(* CODESYS project rmthtc3library.library
   Company: RMTH GmbH
   Title: RMTH TC3 Library
   Placeholder: RMTH TC3 Library
   Version: 1.7

Project tree, tasks and I/O mapping:
  libraries: Tc2_Drive, * (Beckhoff Automation GmbH); Tc2_EtherCAT, * (Beckhoff Automation GmbH); Tc2_MC2, * (Beckhoff Automation GmbH); Tc2_MC2_Drive, * (Beckhoff Automation GmbH); Tc2_NC, * (Beckhoff Automation GmbH); Tc2_Standard, * (Beckhoff Automation GmbH); Tc2_System, * (Beckhoff Automation GmbH); Tc2_Utilities, * (Beckhoff Automation GmbH); Tc3_Interfaces, * (Beckhoff Automation GmbH); Tc3_Module, * (Beckhoff Automation GmbH)
  Configuration/
    Log/
      data type E_LoggingProvider
      data type E_LogLevel
      data type ST_LoggingConfig
    Motion/
      data type E_AxisType
      data type E_EncoderType
  Motion/
    AX5000Diag/
      Structs/
        data type ST_AX5000Diag
      function block FB_AX5000Diag [ST]: A_GetDiagnosis, A_GetDriveRef, A_Reset
    Functions/
      Lenze_84xx/
        function F_DecodeLenze84Status [ST]
    Lenze_84xx/
      function block FB_Antrieb84xxSimple [ST]: A_CalcPosition, A_CheckLatchState, A_Error, A_Test, LatchObjState, Reset
    LenzeIndraDiag/
      Structs/
        data type ST_IndraDriveDiag
      function block FB_IndraDriveDiag [ST]: A_GetDiagnosis, A_GetDriveRef, A_Reset
    MotionCore/
      Enumerations/
        data type E_Mc2AxisState
        data type E_Mc2Cmd
      Structs/
        data type ST_FloatingCmd
        data type ST_FromMc2
        data type ST_Mc2Home
        data type ST_Mc2Jog
        data type ST_Mc2Mov
        data type ST_Mc2SetPos
        data type ST_ToMc2
      function block FB_MC2AXIS [ST]: A_AxisDiag, A_GetCommand, A_Halt, A_Home, A_Jog, A_MovAbs, A_MovAdd, A_MovMod, A_MovRel, A_MovVel, A_Power, A_ResMovExecute, A_SetPosition, A_Stop, A_Tourque
    Structures/
      Lenze_84xx/
        data type IO_84_Lenze_FW2x
        data type ST_84_Lenze_to_PLC
        data type ST_84_PLC_to_Lenze
        data type ST_84_Status
  Utilities/
    Balluff/
      function F_GetBalluffWegValue [ST]
    Enumerations/
      data type E_Direction
      data type E_OperationResult
      data type E_ValveType
    Log/
      Base/
        function block FB_LoggingProviderBase [ST]: AddLog, Run
      Interface/
        interface ITFLoggingProvider: AddLog, Run
      Structures/
        data type ST_Log
      function block FB_DebugLoggingProvider [ST]
      function block FB_EventLoggingProvider [ST]: EventLog, Logger, Run
      function block FB_FileLoggingProvider [ST]: Initialize, Logger, Run, WriteFile
    Math/
      function F_GrayCodeToDecimal [ST]
    StringFunctions/
      StringFunctions/
        function Concat10 [ST]
        function Concat2 [ST]
        function Concat3 [ST]
        function Concat4 [ST]
        function Concat5 [ST]
        function Concat6 [ST]
        function Concat7 [ST]
        function Concat8 [ST]
        function Concat9 [ST]
        function ConcatArray [ST]
        function block FB_GetTimeString [ST]: TimeString
    Structures/
      data type ST_HexColor
    System/
      function F_GetAdsPort [ST]
      function F_GetPlcCycleTime [ST]
      function F_GetSystemTime64 [ST]
      program P_FilePath [ST]
      program P_System [ST]
      data type ST_DefaultPulse
      data type ST_PlcSystemInfo
    function block FB_AsyncDrive [ST]: MoveNeg, MovePos, Reset, Stop
    function block FB_Cylinder [ST]: A_Supervision
    function block FB_CylinderEx [ST]: A_CheckLatchState, A_Supervision, ClearOuts, GoHP, GoWP, LatchObjState, Reset, ResetInit
    function block FB_Pulse [ST]
    function block FB_RotaryEncoder [ST]
    function block FB_ScaleAnalogInput [ST]
    function block FB_Sensor [ST]
    function block FB_TON_RMTH [ST]
  Version/
    global variables Global_Version
  global variables Statics
  global variables StaticsConstant
*)

// Configuration/Log/E_LoggingProvider
TYPE E_LoggingProvider :
(
	///kein Loggingprovider
	eLoggingProviderNone := 0,
	///Filesystem-Loggingprovider
	eLoggingProviderFile := 1,
	///Datenbank-Loggingprovider
	eLoggingProviderDataBase := 2,
	///EventLog-Loggingprovider
	eLoggingProviderEventLog := 3,
	eLoggingProviderNetSvc := 4
);
END_TYPE

// Configuration/Log/E_LogLevel
TYPE E_LogLevel :
(
	///kein Loglevel (nichts wird geloggt)
	eLogLevelNone := 0,
	///nur Fehler werden geloggt
	eLogLevelError := 1,
	///Fehler und Warnungen werden geloggt
	eLogLevelWarning := 2,
	///Fehler, Warnungen und Informationen werden geloggt
	eLogLevelInformation := 3
);
END_TYPE

// Configuration/Log/ST_LoggingConfig
TYPE ST_LoggingConfig :
STRUCT
	/// <info>Angabe des Loggingproviders</info>
	eLoggingProvider: E_LoggingProvider;
	/// <info>Logging Name</info>
	sLogName: STRING;
	/// <info>Logging Pfad</info>
	sLogPath: STRING;
	/// <info>Logging Level</info>
	eLogLevel: E_LogLevel;
END_STRUCT
END_TYPE

// Configuration/Motion/E_AxisType
TYPE E_AxisType :
(
	///	AX5000 hardware	
	AX5xxx,
	///	AX2000 hardware	
	AX2xxx,
	///	EtherCAT Servoterminal		
	EL72xx,
	///	keine HW	
	Virtual,
	///	Digitale IO	
	DigIO,
	///	Lenze 94xx Serie Cia402	
	Lenze_94xx,
	/// Bosch Indradrive EtherCAT
	Bosch_IndradriveEc
);
END_TYPE

// Configuration/Motion/E_EncoderType
TYPE E_EncoderType :
(
	///	kein Feedback	
	None,
	///	Resolver		
	Resolver,
	///	Multiturn Absolute	
	MultiTurnAbs,
	///	Singleturn Absolute	
	SingleTurnAbs
);
END_TYPE

// Motion/AX5000Diag/Structs/ST_AX5000Diag
TYPE ST_AX5000Diag :
STRUCT
	/// NC-Status 
	nNCAxisID: UDINT;
	bOperational: BOOL;
	bC1DError: BOOL;
	bWcStateError: BOOL;
	bAxisError: BOOL;
	iAxisErrorCode: UDINT;
	/// Drive Diag 
	strDriveType: STRING(19);
	strMotorType: STRING(31);
	wDriveStatus: WORD;
	wClass1Diag: WORD;
	stClass1Diag: ST_AX5000_C1D;
	stDriveStatus: ST_AX5000DriveStatus;
	stEcSlaveStateBits: ST_EcSlaveStateBits;
	stEcSlaveState: ST_EcSlaveState;
	bPreopToSafeOpError: BOOL;
	bSafeOpToOpError: BOOL;
	stCPxInvParamList: ST_SoE_CPxInvParamList;
	iDiagNumber: UDINT;
	stDiagNumberList: ST_SoE_DiagNumList;
	strDiagMessage: STRING(19);
END_STRUCT
END_TYPE

// Motion/LenzeIndraDiag/Structs/ST_IndraDriveDiag
TYPE ST_IndraDriveDiag :
STRUCT
	(* NC-Status *)
	nNCAxisID				: UDINT;
	bOperational			: BOOL;
	bC1DError				: BOOL;
	bWcStateError			: BOOL;
	bAxisError				: BOOL;
	iAxisErrorCode			: UDINT;

	(* Drive Diag *)
	strDriveType			: STRING(40);
	strMotorType			: STRING(80);
	wDriveStatus			: WORD;
	wClass1Diag				: WORD;
	stClass1Diag			: ST_IndraDriveCs_C1D;
	stDriveStatus			: ST_IndraDriveCsDriveStatus;
	stEcSlaveStateBits		: ST_EcSlaveStateBits;
	stEcSlaveState			: ST_EcSlaveState;
	bPreopToSafeOpError		: BOOL;
	bSafeOpToOpError		: BOOL;
	stCPxInvParamList		: ST_SoE_CPxInvParamList25;
	iDiagNumber				: UDINT;
	stDiagNumberList		: ST_SoE_DiagNumList50;
	strDiagMessage			: STRING(80);	
END_STRUCT
END_TYPE

// Motion/MotionCore/Enumerations/E_Mc2AxisState
TYPE E_Mc2AxisState :
(
	Mc2AxisStateInit,
	Mc2AxisStateIdle,
	Mc2AxisStateEnable,
	Mc2AxisStateDisable,
	Mc2AxisStateHome,
	Mc2AxisStateHalt,
	Mc2AxisStateStop,
	Mc2AxisStateSetPos,
	Mc2AxisStateJog,
	Mc2AxisStateMovAbs,
	Mc2AxisStateMovRel,
	Mc2AxisStateMovAdd,
	Mc2AxisStateMovMod,
	Mc2AxisStateMovVel,
	Mc2AxisStateError,
	Mc2AxisStateReset
);
END_TYPE

// Motion/MotionCore/Enumerations/E_Mc2Cmd
TYPE E_Mc2Cmd :
(
	Mc2CmdNothing,
	Mc2CmdSetPos,
	///	homing				
	Mc2CmdHome,
	///	normal stop			
	Mc2CmdHalt,
	///	stop with restart lock	
	Mc2CmdStop,
	Mc2CmdJog,
	Mc2CmdMovAbs,
	Mc2CmdMovRel,
	Mc2CmdMovAdd,
	Mc2CmdMovMod,
	Mc2CmdMovVel,
	Mc2CmdReset
);
END_TYPE

// Motion/MotionCore/Structs/ST_FloatingCmd
TYPE ST_FloatingCmd :
STRUCT
	///	Schwimmend EIN	
	bFloatingOn: BOOL;
	///	in Richtung drücken	
	bPush: BOOL;
	///	Weg für Drücken	
	fPushPos: REAL := -0.1;
	///	Speed für Drücken	
	fPushVel: REAL := 1;
END_STRUCT
END_TYPE

// Motion/MotionCore/Structs/ST_FromMc2
TYPE ST_FromMc2 :
STRUCT
	nAxisId: DWORD;
	AxisState: E_Mc2AxisState;
	sStatusText: STRING;
	bEnabled: BOOL;
	bError: BOOL;
	sErrorSource: STRING(80);
	nErrorId: UDINT;
	///	actual Pos	
	fActPos: REAL;
	///	actual modulo pos	
	fActModPos: REAL;
	///	aktuelles Drehmoment -> 0..100 % von Antriebseinstellung	
	fActMoment: REAL;
	///	aktuelle Geschwindigkeit	
	fActVelo: REAL;
	bNotMoving: BOOL;
	///	Achse fährt Positive Richtung	
	bMovesPos: BOOL;
	///	Achse fährt Negative Richtung	
	bMovesNeg: BOOL;
	///	Achse hat Auftrag, führt Auftrag aus	
	bHasJob: BOOL;
	bReady: BOOL;
	InTargetPosition: BOOL;
	bCoupled: BOOL;
	///	Power function block output data 		
	PowerAxisOut: ST_McOutputs;
	///	Reset function block output data 		
	ResetOut: ST_McOutputs;
	///	Home function block output data		
	HomeOut: ST_McOutputs;
	///	MoveAbs function block output data 	
	MoveAbsOut: ST_McOutputs;
	MoveAbsOut1: ST_McOutputs;
	MoveAbsOut2: ST_McOutputs;
	///	MoveRel function block output data	
	MoveRelOut: ST_McOutputs;
	MoveRelOut1: ST_McOutputs;
	MoveRelOut2: ST_McOutputs;
	///	MoveAddfunction block output data	
	MoveAddOut: ST_McOutputs;
	MoveAddOut1: ST_McOutputs;
	MoveAddOut2: ST_McOutputs;
	///	MoveVel function block output data	
	MoveVelOut: ST_McOutputs;
	MoveVelOut1: ST_McOutputs;
	MoveVelOut2: ST_McOutputs;
	///	Jog function block output data 	
	JogOut: ST_McOutputs;
	///	MoveMod function block output data 	
	MoveModOut: ST_McOutputs;
	///	StopOut function block output data	
	StopOut: ST_McOutputs;
	///	HaltOutfunction block output data		
	HaltOut: ST_McOutputs;
END_STRUCT
END_TYPE

// Motion/MotionCore/Structs/ST_Mc2Home
TYPE ST_Mc2Home :
STRUCT
	Position: LREAL := DEFAULT_HOME_POSITION;
	HomingMode: MC_HomingMode := MC_DefaultHoming;
	BufferMode: MC_BufferMode;
END_STRUCT
END_TYPE

// Motion/MotionCore/Structs/ST_Mc2Jog
TYPE ST_Mc2Jog :
STRUCT
	JogForward: BOOL;
	JogBackwards: BOOL;
	Mode: E_JogMode;
	Position: LREAL;
	Velocity: LREAL;
	Acceleration: LREAL;
	Deceleration: LREAL;
	Jerk: LREAL;
END_STRUCT
END_TYPE

// Motion/MotionCore/Structs/ST_Mc2Mov
TYPE ST_Mc2Mov :
STRUCT
	Position: LREAL;
	Velocity: LREAL;
	Acceleration: LREAL;
	Deceleration: LREAL;
	Jerk: LREAL;
	BufferMode: MC_BufferMode := MC_Aborting;
	Direction: MC_Direction;
END_STRUCT
END_TYPE

// Motion/MotionCore/Structs/ST_Mc2SetPos
TYPE ST_Mc2SetPos :
STRUCT
	Position: LREAL;
	///	Die Achsposition wird auf einen absoluten Wert gesetzt, wenn Mode=FALSE ist. Anderenfalls wird die Achsposition relativ um den angegebenen Wert Position verändert. 	
	Mode: BOOL;
	///	ClearPositionLag kann optional gesetzt werden, falls Soll- und Istposition auf den gleichen Wert gesetzt werden sollen. Damit wird der Schleppfehler gelöscht.	
	ClearPositionLag: BOOL := FALSE;
END_STRUCT
END_TYPE

// Motion/MotionCore/Structs/ST_ToMc2
TYPE ST_ToMc2 :
STRUCT
	Command: E_Mc2Cmd;
	strctJogPrm: ST_Mc2Jog;
	strctMovPrm: ST_Mc2Mov;
	strctHomPrm: ST_Mc2Home;
	strctSetPosPrm: ST_Mc2SetPos;
END_STRUCT
END_TYPE

// Motion/Structures/Lenze_84xx/IO_84_Lenze_FW2x
TYPE IO_84_Lenze_FW2x :
STRUCT
	wStatus_Control			: WORD ;	(*W1*)
	wIn02					: INT ;
	wIn03					: INT ;
	wIn04					: INT ;
	wIn05					: INT ;
	wIn06					: INT ;
	wIn07					: INT ;
	wIn08					: INT ;
	wIn09					: INT ;
	wIn10					: INT ;
	wIn11					: INT ;
	wIn12					: INT ;
	wIn13					: INT ;
	wIn14					: INT ;
	wIn15					: INT ;
	wIn16					: INT ;
END_STRUCT
END_TYPE

// Motion/Structures/Lenze_84xx/ST_84_Lenze_to_PLC
TYPE ST_84_Lenze_to_PLC :
STRUCT
	wStatus					: WORD ;	(*W1*)
	nIstDrz					: INT ;	(*W2*)
	nResolverPos			: DINT ;	(* W3 u 4*)
	nMotTemperatur			: INT ;		(*W5*)
	nIstMom					: INT ;	(* W6*)
	nRotPos					: INT ;		(*W7*)

(* 	Zur SPS vom Regler:

W1 Statuswort New
Bit0		Drive Ready
Bit1		Impulssperre (gesperrt von SPS)
Bit2		free
Bit3		free
Bit4		free
Bit5		free
Bit6		Aktuelle Drehzahl < C24 (Moving..)
Bit7		Reglersperre aktiv
Bit8		ZustandsID Bit 0
Bit9		ZustandsID Bit 1
Bit10 	ZustandsID Bit 2
Bit11 	ZustandsID Bit 3
Bit12 	Warning aktiv
Bit13 	Fail aktiv
Bit14 	free
Bit15 	Motor über Temperatur Grenze	

	über Codierung Bit 8-11
	Drive Operation enabled
	QSP aktiv
	Drive ready to switch on	(	Bit 8 = 1, Bit 9 = 1, Bit 10 = 0, Bit 11 = 0	)
	-
	- Unterspannung Zwischenkreis -> nicht vorhanden
	- Reglersperre 9400 durch Engineer freizugeben ! -> Reglersperre aktiv

W2 Istdrehzahl
(100% == xxx rpm == 2^14 == 16384) xxx = Bezugsdrehzahl

W3 und W4 Resolverposition
(2^16 / U == ??? == ??? umdr)

W5 Motortemperatur
(200 == 200°C)

W6 Istdrehmoment
(100% == xx Nm == 2^14 == 16384)

W6 Rotorposition (ungenau, 20ms)
(2048 / U)

*)
END_STRUCT
END_TYPE

// Motion/Structures/Lenze_84xx/ST_84_PLC_to_Lenze
TYPE ST_84_PLC_to_Lenze :
STRUCT
	wControl				: WORD ;
	nSollDrz					: INT ;
	nMaxMom				: INT ;		(* 2^14 = 100% *)
	nGWMotTempLuefter	: INT ;
	nReseve				: INT ;

(* 	Von SPS zum Regler

W1 Controlwort New
Bit0		Drive Switch ON (ON nach Sperre)
Bit1		Impulssperre 
Bit2		QSP
Bit3		RFR (Reglerfreigabe mit high)
Bit4		
Bit5		
Bit6	
Bit7		Trip Reset (Fehlerreset)
Bit8		Break release (wenn händisch gelöst werden will - wird sonst durch RFR autom. in Antrieb erledigt)*
Bit9		free
Bit10 	free
Bit11 	free
Bit12 	Jog1
Bit13 	free
Bit14 	free
Bit15 	Drehrichtungsumkehr	

Speed follower enable ist bei 84er immer wenn Applikation "Geschwindigkeitsregelung" - Stellantrieb Drehzahl

W2 Solldrehzahl
(100% == xxx rpm == 16384 == 2^14)

W3 Maximaldrehmoment
(100% == xxx Nm == 16384 == 2^14)

W4 Solltemperatur für Lüfter Ein
(200 == 200°C)

ab W5 Reserve
*)
END_STRUCT
END_TYPE

// Motion/Structures/Lenze_84xx/ST_84_Status
TYPE ST_84_Status :
STRUCT
	bDriveReady				:BOOL;	(*	Drive Ready to Move	*)
	bImpulssperre			:BOOL;	(*	Impulssperre (gesperrt von SPS)	*)
	bNotMoving				:BOOL;
	bReglersperreAktiv		:BOOL;
	bDriveReadyToSwitchOn	:BOOL;
	bDriveOperationEnabled	:BOOL;
	bQSPAktiv				:BOOL;
	bWarningAktiv			:BOOL;	(*	Bit12 	Warning aktiv		*)
	bFailAktiv				:BOOL;	(*	Bit13 	Fail aktiv		*)
	bMotorTempHigh			:BOOL;

(* 	Zur SPS vom Regler:

W1 Statuswort New
Bit0		Drive Ready
Bit1		Impulssperre (gesperrt von SPS)
Bit2		free
Bit3		free
Bit4		free
Bit5		free
Bit6		Aktuelle Drehzahl < C24 (Moving..)
Bit7		Reglersperre aktiv
Bit8		ZustandsID Bit 0
Bit9		ZustandsID Bit 1
Bit10 	ZustandsID Bit 2
Bit11 	ZustandsID Bit 3
Bit12 	Warning aktiv
Bit13 	Fail aktiv
Bit14 	free
Bit15 	Motor über Temperatur Grenze	

	über Codierung Bit 8-11
	Drive Operation enabled
	QSP aktiv
	Drive ready to switch on	(	Bit 8 = 1, Bit 9 = 1, Bit 10 = 0, Bit 11 = 0	)
	-
	- Unterspannung Zwischenkreis -> nicht vorhanden
	- Reglersperre 9400 durch Engineer freizugeben ! -> Reglersperre aktiv

W2 Istdrehzahl
(100% == 1455rpm == 2^15) (30)

W3 Istdrehmoment
(Abhaspel: 100% == 82,13Nm == 2^15) (30)
(Aufhaspel: 100% == Nm == 2^15) (30)

W4 Rotorposition
(10000 == 360° == 1 umdr )

W5 Motortemperatur
(200 == 200°C)

W6 Reserve (Rotorlage von Codestelle C60 ausgelesen)
(0 bis 2047 == eine Motorumdrehung)
*)
END_STRUCT
END_TYPE

// Utilities/Enumerations/E_Direction
TYPE E_Direction :
(
	NODIRECTION,
	FORWARD,
	BACKWARD
);
END_TYPE

// Utilities/Enumerations/E_OperationResult
/// Enumeration of possible op results
TYPE E_OperationResult :
(
	/// operation result not initialized
	eOperationResult_None := 0,
	/// operation process busy
	eOperationResult_Busy,
	/// operation succeeded or true
	eOperationResult_Ok,
	/// operation result not ok or false
	eOperationResult_NOk,
	/// operation failed/error
	eOperationResult_Error
);
END_TYPE

// Utilities/Enumerations/E_ValveType
TYPE E_ValveType :
(
	/// 5/2 Wege, bistabil
	eValvetype_Default := 0,
	/// 5/2 Wege, bistabil
	eValvetype_5_2_bi := 1,
	/// 3/2 Wege, federrueckstellend
	eValvetype_3_2_mono := 2,
	/// 5/3 Wege, Mittelstellung gesperrt
	eValvetype_5_3_lock := 3,
	/// 5/3 Wege, Mittelstellung drucklos
	eValvetype_5_3_unlock := 4
);
END_TYPE

// Utilities/Log/Structures/ST_Log
TYPE ST_Log :
STRUCT
	sText: T_MaxString;
	sSource: STRING;
	bSaveRequest: BOOL;
	bSaved: BOOL;
	///	eLogLevelNone, eLogLevelError, eLogLevelWarning, eLogLevelInformation	
	eLevel: E_LogLevel;
	sTime: STRING;
END_STRUCT
END_TYPE

// Utilities/Structures/ST_HexColor
//	Color Hexcode...[generiert aus .net]
TYPE ST_HexColor :
STRUCT
	ActiveBorder :DINT:=16#D4D0C8;
	ActiveCaption :DINT:=16#0054E3;
	ActiveCaptionText :DINT:=16#FFFFFF;
	AliceBlue :DINT:=16#F0F8FF;
	AntiqueWhite :DINT:=16#FAEBD7;
	AppWorkspace :DINT:=16#808080;
	Aqua :DINT:=16#00FFFF;
	Aquamarine :DINT:=16#7FFFD4;
	Azure :DINT:=16#F0FFFF;
	Beige :DINT:=16#F5F5DC;
	Bisque :DINT:=16#FFE4C4;
	Black :DINT:=16#000000;
	BlanchedAlmond :DINT:=16#FFEBCD;
	Blue :DINT:=16#0000FF;
	BlueViolet :DINT:=16#8A2BE2;
	Brown :DINT:=16#A52A2A;
	BurlyWood :DINT:=16#DEB887;
	ButtonFace :DINT:=16#ECE9D8;
	ButtonHighlight :DINT:=16#FFFFFF;
	ButtonShadow :DINT:=16#ACA899;
	CadetBlue :DINT:=16#5F9EA0;
	Chartreuse :DINT:=16#7FFF00;
	Chocolate :DINT:=16#D2691E;
	Control :DINT:=16#ECE9D8;
	ControlDark :DINT:=16#ACA899;
	ControlDarkDark :DINT:=16#716F64;
	ControlLight :DINT:=16#F1EFE2;
	ControlLightLight :DINT:=16#FFFFFF;
	ControlText :DINT:=16#000000;
	Coral :DINT:=16#FF7F50;
	CornflowerBlue :DINT:=16#6495ED;
	Cornsilk :DINT:=16#FFF8DC;
	Crimson :DINT:=16#DC143C;
	Cyan :DINT:=16#00FFFF;
	DarkBlue :DINT:=16#00008B;
	DarkCyan :DINT:=16#008B8B;
	DarkGoldenrod :DINT:=16#B8860B;
	DarkGray :DINT:=16#A9A9A9;
	DarkGreen :DINT:=16#006400;
	DarkKhaki :DINT:=16#BDB76B;
	DarkMagenta :DINT:=16#8B008B;
	DarkOliveGreen :DINT:=16#556B2F;
	DarkOrange :DINT:=16#FF8C00;
	DarkOrchid :DINT:=16#9932CC;
	DarkRed :DINT:=16#8B0000;
	DarkSalmon :DINT:=16#E9967A;
	DarkSeaGreen :DINT:=16#8FBC8B;
	DarkSlateBlue :DINT:=16#483D8B;
	DarkSlateGray :DINT:=16#2F4F4F;
	DarkTurquoise :DINT:=16#00CED1;
	DarkViolet :DINT:=16#9400D3;
	DeepPink :DINT:=16#FF1493;
	DeepSkyBlue :DINT:=16#00BFFF;
	Desktop :DINT:=16#004E98;
	DimGray :DINT:=16#696969;
	DodgerBlue :DINT:=16#1E90FF;
	Firebrick :DINT:=16#B22222;
	FloralWhite :DINT:=16#FFFAF0;
	ForestGreen :DINT:=16#228B22;
	Fuchsia :DINT:=16#FF00FF;
	Gainsboro :DINT:=16#DCDCDC;
	GhostWhite :DINT:=16#F8F8FF;
	Gold :DINT:=16#FFD700;
	Goldenrod :DINT:=16#DAA520;
	GradientActiveCaption :DINT:=16#3D95FF;
	GradientInactiveCaption :DINT:=16#9DB9EB;
	Gray :DINT:=16#808080;
	GrayText :DINT:=16#ACA899;
	Green :DINT:=16#008000;
	GreenYellow :DINT:=16#ADFF2F;
	Highlight :DINT:=16#316AC5;
	HighlightText :DINT:=16#FFFFFF;
	Honeydew :DINT:=16#F0FFF0;
	HotPink :DINT:=16#FF69B4;
	HotTrack :DINT:=16#000080;
	InactiveBorder :DINT:=16#D4D0C8;
	InactiveCaption :DINT:=16#7A96DF;
	InactiveCaptionText :DINT:=16#D8E4F8;
	IndianRed :DINT:=16#CD5C5C;
	Indigo :DINT:=16#4B0082;
	Info :DINT:=16#FFFFE1;
	InfoText :DINT:=16#000000;
	Ivory :DINT:=16#FFFFF0;
	Khaki :DINT:=16#F0E68C;
	Lavender :DINT:=16#E6E6FA;
	LavenderBlush :DINT:=16#FFF0F5;
	LawnGreen :DINT:=16#7CFC00;
	LemonChiffon :DINT:=16#FFFACD;
	LightBlue :DINT:=16#ADD8E6;
	LightCoral :DINT:=16#F08080;
	LightCyan :DINT:=16#E0FFFF;
	LightGoldenrodYellow :DINT:=16#FAFAD2;
	LightGray :DINT:=16#D3D3D3;
	LightGreen :DINT:=16#90EE90;
	LightPink :DINT:=16#FFB6C1;
	LightSalmon :DINT:=16#FFA07A;
	LightSeaGreen :DINT:=16#20B2AA;
	LightSkyBlue :DINT:=16#87CEFA;
	LightSlateGray :DINT:=16#778899;
	LightSteelBlue :DINT:=16#B0C4DE;
	LightYellow :DINT:=16#FFFFE0;
	Lime :DINT:=16#00FF00;
	LimeGreen :DINT:=16#32CD32;
	Linen :DINT:=16#FAF0E6;
	Magenta :DINT:=16#FF00FF;
	Maroon :DINT:=16#800000;
	MediumAquamarine :DINT:=16#66CDAA;
	MediumBlue :DINT:=16#0000CD;
	MediumOrchid :DINT:=16#BA55D3;
	MediumPurple :DINT:=16#9370DB;
	MediumSeaGreen :DINT:=16#3CB371;
	MediumSlateBlue :DINT:=16#7B68EE;
	MediumSpringGreen :DINT:=16#00FA9A;
	MediumTurquoise :DINT:=16#48D1CC;
	MediumVioletRed :DINT:=16#C71585;
	Menu :DINT:=16#FFFFFF;
	MenuBar :DINT:=16#ECE9D8;
	MenuHighlight :DINT:=16#316AC5;
	MenuText :DINT:=16#000000;
	MidnightBlue :DINT:=16#191970;
	MintCream :DINT:=16#F5FFFA;
	MistyRose :DINT:=16#FFE4E1;
	Moccasin :DINT:=16#FFE4B5;
	NavajoWhite :DINT:=16#FFDEAD;
	Navy :DINT:=16#000080;
	OldLace :DINT:=16#FDF5E6;
	Olive :DINT:=16#808000;
	OliveDrab :DINT:=16#6B8E23;
	Orange :DINT:=16#FFA500;
	OrangeRed :DINT:=16#FF4500;
	Orchid :DINT:=16#DA70D6;
	PaleGoldenrod :DINT:=16#EEE8AA;
	PaleGreen :DINT:=16#98FB98;
	PaleTurquoise :DINT:=16#AFEEEE;
	PaleVioletRed :DINT:=16#DB7093;
	PapayaWhip :DINT:=16#FFEFD5;
	PeachPuff :DINT:=16#FFDAB9;
	Peru :DINT:=16#CD853F;
	Pink :DINT:=16#FFC0CB;
	Plum :DINT:=16#DDA0DD;
	PowderBlue :DINT:=16#B0E0E6;
	Purple :DINT:=16#800080;
	Red :DINT:=16#FF0000;
	RosyBrown :DINT:=16#BC8F8F;
	RoyalBlue :DINT:=16#4169E1;
	SaddleBrown :DINT:=16#8B4513;
	Salmon :DINT:=16#FA8072;
	SandyBrown :DINT:=16#F4A460;
	ScrollBar :DINT:=16#D4D0C8;
	SeaGreen :DINT:=16#2E8B57;
	SeaShell :DINT:=16#FFF5EE;
	Sienna :DINT:=16#A0522D;
	Silver :DINT:=16#C0C0C0;
	SkyBlue :DINT:=16#87CEEB;
	SlateBlue :DINT:=16#6A5ACD;
	SlateGray :DINT:=16#708090;
	Snow :DINT:=16#FFFAFA;
	SpringGreen :DINT:=16#00FF7F;
	SteelBlue :DINT:=16#4682B4;
	TTAN :DINT:=16#D2B48C;
	Teal :DINT:=16#008080;
	Thistle :DINT:=16#D8BFD8;
	Tomato :DINT:=16#FF6347;
	Transparent :DINT:=16#FFFFFF;
	Turquoise :DINT:=16#40E0D0;
	Violet :DINT:=16#EE82EE;
	Wheat :DINT:=16#F5DEB3;
	White :DINT:=16#FFFFFF;
	WhiteSmoke :DINT:=16#F5F5F5;
	Window :DINT:=16#FFFFFF;
	WindowFrame :DINT:=16#000000;
	WindowText :DINT:=16#000000;
	Yellow :DINT:=16#FFFF00;
	YellowGreen :DINT:=16#9ACD32;
END_STRUCT
END_TYPE

// Utilities/System/ST_DefaultPulse
TYPE ST_DefaultPulse :
STRUCT
	/// default impulse flags
	bImpulse1000ms: BOOL;
	bImpulse500ms: BOOL;
	bImpulse300ms: BOOL;
	bImpulse200ms: BOOL;
	bImpulse100ms: BOOL;
	/// default toggle flags
	bToggle1000ms: BOOL;
	bToggle500ms: BOOL;
	bToggle300ms: BOOL;
	bToggle200ms: BOOL;
	bToggle100ms: BOOL;
END_STRUCT
END_TYPE

// Utilities/System/ST_PlcSystemInfo
TYPE ST_PlcSystemInfo :
STRUCT
	/// system info structure
	stPlcAppSystemInfo: PlcAppSystemInfo;
	/// tast info structure
	stPlcTaskSystemInfo: PlcTaskSystemInfo;
	/// cycle time from task configuration in [s]
	fCycleTime: LREAL;
	/// needed cycletime for the last cycle in [s]
	fLastExecTime: LREAL;
END_STRUCT
END_TYPE

// Version/Global_Version
// This function has been automatically generated from the project information.
VAR_GLOBAL CONSTANT
	{attribute 'const_non_replaced'}
	stLibVersion_RMTH_TC3_Library : ST_LibVersion := (iMajor := 1, iMinor := 7, iBuild := 0, iRevision := 0, sVersion := '1.7');
END_VAR

// Statics
VAR_GLOBAL
	/// current system time
	dtNow: DT;
	/// current system time in string format	
	sTimeString: STRING;
	/// PLC system informations
	stPlcSystemInfo: ST_PlcSystemInfo;
	/// default pulse struct
	stPulse: ST_DefaultPulse;
	/// colors
	stColor: ST_HexColor;
	/// logging buffer
	arLoggs: ARRAY[0..iLogArraySize] OF ST_Log;
	/// global stuff
	bForceStateChgAfterDrvReset: BOOL;
	bLogDriveDiagMsgs: BOOL;
END_VAR

// StaticsConstant
VAR_GLOBAL CONSTANT
	sEmpty: STRING(0) := '';
	dtMinValue: DT := DATE_AND_TIME#1970-1-1-0:0;
	dtMaxValue: DT := DATE_AND_TIME#2106-2-6-6:28:15;
	iLogArraySize: INT := 500;
END_VAR

// Motion/AX5000Diag/FB_AX5000Diag
FUNCTION_BLOCK FB_AX5000Diag
VAR_INPUT
	/// AmsNetId of the IPC 
	IPCNetID: T_AmsNetId;
	Timeout: TIME := DEFAULT_ADS_TIMEOUT;
	Reset: BOOL;
	GetDiag: BOOL;
END_VAR
VAR_IN_OUT
	Axis: AXIS_REF;
	stAX5000Diag: ST_AX5000Diag;
END_VAR
VAR_OUTPUT
	Error: BOOL;
	AdsErrId: UINT;
	SercosErrId: UINT;
	ResetAct: BOOL;
	ResetDone: BOOL;
	DiagAct: BOOL;
	Busy: BOOL;
	/// contains sNetID of EcMaster, nSlaveAddr of EcDrive, nDriveNo of EcDrive, either preset or read from NC 
	DriveRef: ST_DriveRef;
END_VAR
VAR
	iState: INT;
	iSubState: INT;
	GetDriveRef: BOOL := TRUE;
	AxisID: UDINT;
	C1DErrorPrev: BOOL;
	WcStateErrorPrev: BOOL;
	AxisErrorPrev: BOOL;
	OperationalPrev: BOOL;
	ResetPrev: BOOL;
	GetDiagPrev: BOOL;
	fbSoERead: FB_SoERead;
	fbDiagMessage: FB_SoEReadDiagMessage;
	fbClassXDiag: FB_SoEReadClassXDiag;
	fbDiagNumber: FB_SoEReadDiagNumber;
	fbDiagNumberList: FB_SoEReadDiagNumberList;
	fbReset: FB_SoEReset;
	fbDelay: TON;
	fbGetSlaveState: FB_EcGetSlaveState;
	fbReqSlaveState: FB_EcReqSlaveState;
	fbNcReset: MC_Reset;
	fbAdsRead: ADSREAD;
	readBuffer: ARRAY[0..9] OF BYTE;
	Ids: T_AmsNetIdArr;
	fbFormatString: FB_FormatString;
	DiagMsgPrev: STRING(255);
	LogMsg: STRING(255);
	strSoEString: ST_SoE_StringEx;
	I: INT;
END_VAR
VAR CONSTANT
	/// Axis with ID: Parameter 			
	NCIDXG_AXPARMS: UDINT := 16#4000;
	NCIDXO_AXP_HWAMSADDR: UDINT := 16#31;
END_VAR

stAX5000Diag.bOperational	:= Axis.NcToPlc.StateDWord.0;
stAX5000Diag.bC1DError	 	:= Axis.NcToPlc.StateDWord.28;
stAX5000Diag.bWcStateError 	:= Axis.NcToPlc.StateDWord.30;
stAX5000Diag.bAxisError		:= Axis.NcToPlc.StateDWord.31;
stAX5000Diag.iAxisErrorCode	:= Axis.NcToPlc.ErrorCode;

CASE iState OF
0:	(* idle *)
	GetDriveRef 	:= (DriveRef.nSlaveAddr = 0);

	IF GetDriveRef THEN
		Busy			:= TRUE;
		Error			:= FALSE;
		AdsErrId		:= 0;
		SercosErrId		:= 0;
		iState 			:= 1;
		iSubState		:= 0;
		AxisID 			:= Axis.NcToPlc.AxisId;

	ELSIF Reset AND NOT ResetPrev THEN
		Busy			:= TRUE;
		ResetAct			:= TRUE;
		ResetPrev		:= Reset;
		Error			:= FALSE;
		AdsErrId			:= 0;
		SercosErrId		:= 0;
		iState 			:= 2;
		iSubState		:= 0;
		AxisID 			:= Axis.NcToPlc.AxisId;

	ELSIF GetDiag AND NOT GetDiagPrev OR
		(stAX5000Diag.bC1DError AND NOT C1DErrorPrev) OR (NOT stAX5000Diag.bC1DError AND C1DErrorPrev) (* rising/falling C1D *) OR
		(stAX5000Diag.bWcStateError AND NOT WcStateErrorPrev) OR (NOT stAX5000Diag.bWcStateError AND WcStateErrorPrev) (* rising/falling WcState *) OR
		(stAX5000Diag.bAxisError AND NOT AxisErrorPrev) OR (NOT stAX5000Diag.bAxisError AND AxisErrorPrev) (* rising/falling NcError *) OR
		(stAX5000Diag.bOperational AND NOT OperationalPrev) OR (NOT stAX5000Diag.bOperational AND OperationalPrev) (* rising/falling Enable *) THEN

		Busy			:= TRUE;
		DiagAct			:= TRUE;
		GetDiagPrev		:= GetDiag;
		Error			:= FALSE;
		AdsErrId		:= 0;
		SercosErrId		:= 0;
		iState 			:= 3;
		iSubState		:= 0;
		AxisID 			:= Axis.NcToPlc.AxisId;

		(* set/clear flags *)
		C1DErrorPrev		:= stAX5000Diag.bC1DError;
		WcStateErrorPrev	:= stAX5000Diag.bWcStateError;
		AxisErrorPrev		:= stAX5000Diag.bAxisError;
		OperationalPrev		:= stAX5000Diag.bOperational;

	ELSE
		ResetAct		:= FALSE;
		ResetDone 	:= ResetPrev AND (stAX5000Diag.bOperational AND NOT stAX5000Diag.bAxisError);
		DiagAct		:= FALSE;
	END_IF

1:	(* get drive reference *)
	A_GetDriveRef( );

2:	(* reset and state change *)
	A_Reset( );

3:	(* get diag data *)
	A_GetDiagnosis( );

END_CASE

(* clear latch *)
ResetPrev	:= ResetPrev AND Reset;
(*	wenn Fehler -> neuer Reset	*)
IF NOT (stAX5000Diag.bOperational AND NOT stAX5000Diag.bAxisError) THEN
	ResetPrev := FALSE;
END_IF

GetDiagPrev	:= GetDiagPrev AND GetDiag;

ACTION A_GetDiagnosis:

CASE iSubState OF

	0:	fbClassXDiag(
			NetId		:= IPCNetID,
			Execute		:= TRUE,
			DiagClass 	:= 1,
			Timeout		:= DEFAULT_ADS_TIMEOUT,
			Axis		:= Axis,
		);
	
		IF NOT fbClassXDiag.Busy THEN
			fbClassXDiag(Execute:= FALSE,Axis := Axis);
	
			IF NOT fbClassXDiag.Error THEN
				stAX5000Diag.wClass1Diag	:= fbClassXDiag.ClassXDiag;
				stAX5000Diag.stClass1Diag	:= F_ConvWordToSTAX5000C1D(stAX5000Diag.wClass1Diag);
			ELSE
				Error			:= TRUE;
				AdsErrId		:= fbClassXDiag.AdsErrId;
				SercosErrId	:= fbClassXDiag.SercosErrId;
			END_IF
			iSubState	:= iSubState + 1;
		END_IF

	1:	fbDiagMessage(
			NetId	:= IPCNetID,
			Execute	:= TRUE,
			Timeout	:= DEFAULT_ADS_TIMEOUT,
			Axis	:= Axis,
		);
	
		IF NOT fbDiagMessage.Busy THEN
			fbDiagMessage(Execute:= FALSE,Axis := Axis);
	
			IF NOT fbDiagMessage.Error THEN
				stAX5000Diag.strDiagMessage := LEFT(fbDiagMessage.DiagMessage.strData, UINT_TO_INT(fbDiagMessage.DiagMessage.iActualSize));
			ELSE
				Error			:= TRUE;
				AdsErrId		:= fbDiagMessage.AdsErrId;
				SercosErrId	:= fbDiagMessage.SercosErrId;
			END_IF
			iSubState	:= iSubState + 1;
		END_IF
	
	2:	fbDiagNumber(
			NetId	:= IPCNetID,
			Execute	:= TRUE,
			Timeout	:= DEFAULT_ADS_TIMEOUT,
			Axis	:= Axis,
		);
	
		IF NOT fbDiagNumber.Busy THEN
			fbDiagNumber(Execute:= FALSE,Axis := Axis);
	
			IF NOT fbDiagNumber.Error THEN
				stAX5000Diag.iDiagNumber := fbDiagNumber.DiagNumber;
			ELSE
				Error			:= TRUE;
				AdsErrId		:= fbDiagNumber.AdsErrId;
				SercosErrId	:= fbDiagNumber.SercosErrId;
			END_IF
			iSubState	:= iSubState + 1;
		END_IF
	
	3:	fbSoERead(
			NetId	:= IPCNetID,
			Execute	:= TRUE,
			Idn		:= 135,
			Element	:=16#44,
			pDstBuf	:=ADR(stAX5000Diag.wDriveStatus),
			BufLen	:=SIZEOF(stAX5000Diag.wDriveStatus),
			Timeout	:= DEFAULT_ADS_TIMEOUT,
			Axis	:= Axis,
		);
	
		IF NOT fbSoERead.Busy THEN
			fbSoERead(Execute:= FALSE,Axis := Axis);
			IF NOT fbSoERead.Error THEN
				stAX5000Diag.stDriveStatus := F_ConvWordToSTAX5000DriveStatus(stAX5000Diag.wDriveStatus);
				iSubState		:= iSubState + 1;
			ELSE
				Error			:= TRUE;
				AdsErrId		:= fbSoERead.AdsErrId;
				SercosErrId	:= fbSoERead.SercosErrId;
				iSubState		:= iSubState + 2;
			END_IF
		END_IF
	
	4:	fbSoERead(
			NetId	:= IPCNetID,
			Execute	:= TRUE,
			Idn		:= stAX5000Diag.stDriveStatus.iActOpModeParNum,
			Element	:=16#44,
			pDstBuf	:=ADR(stAX5000Diag.stDriveStatus.eActOpMode),
			BufLen	:=SIZEOF(stAX5000Diag.stDriveStatus.eActOpMode),
			Timeout	:= DEFAULT_ADS_TIMEOUT,
			Axis	:= Axis,
		);
	
		IF NOT fbSoERead.Busy THEN
			fbSoERead(Execute:= FALSE,Axis := Axis);
			IF NOT fbSoERead.Error THEN
				;
			ELSE
				Error			:= TRUE;
				AdsErrId		:= fbSoERead.AdsErrId;
				SercosErrId	:= fbSoERead.SercosErrId;
			END_IF
			iSubState	:= iSubState + 1;
		END_IF
	
	5:	fbGetSlaveState(
			sNetId		:= DriveRef.sNetId,
			nSlaveAddr	:= DriveRef.nSlaveAddr,
			bExecute	:= TRUE,
			tTimeout	:= DEFAULT_ADS_TIMEOUT,
		);
	
		IF NOT fbGetSlaveState.bBusy THEN
			fbGetSlaveState(bExecute:= FALSE);
			IF NOT fbGetSlaveState.bError THEN
				stAX5000Diag.stEcSlaveState := fbGetSlaveState.state;
				stAX5000Diag.stEcSlaveStateBits := F_ConvSlaveStateToBits(fbGetSlaveState.state);
			ELSE
				Error			:= TRUE;
				AdsErrId		:= UDINT_TO_UINT(fbGetSlaveState.nErrId);
			END_IF
	
			IF stAX5000Diag.stEcSlaveStateBits.bError THEN
				IF stAX5000Diag.stEcSlaveStateBits.bPreop THEN
					(* read S21 - IDN List of Invalid operation data for CP2 (Preop->SaveOp) *)
					MEMSET(ADR(stAX5000Diag.stCPxInvParamList), 0, SIZEOF(stAX5000Diag.stCPxInvParamList));
					stAX5000Diag.bPreopToSafeOpError := TRUE;
					stAX5000Diag.bSafeOpToOpError := FALSE;
					iSubState	:= iSubState + 1;
				ELSIF stAX5000Diag.stEcSlaveStateBits.bSafeOp THEN
					(* read S22 - IDN List of Invalid operation data for CP3 (SaveOp->Op) *)
					MEMSET(ADR(stAX5000Diag.stCPxInvParamList), 0, SIZEOF(stAX5000Diag.stCPxInvParamList));
					stAX5000Diag.bPreopToSafeOpError := FALSE;
					stAX5000Diag.bSafeOpToOpError := TRUE;
					iSubState	:= iSubState + 2;
				ELSE
					(* Skip S21 + S22 *)
					MEMSET(ADR(stAX5000Diag.stCPxInvParamList), 0, SIZEOF(stAX5000Diag.stCPxInvParamList));
					stAX5000Diag.bPreopToSafeOpError := FALSE;
					stAX5000Diag.bSafeOpToOpError := FALSE;
					iSubState	:= iSubState + 3;
				END_IF
			ELSE
				(* Skip S21 + S22 *)
				MEMSET(ADR(stAX5000Diag.stCPxInvParamList), 0, SIZEOF(stAX5000Diag.stCPxInvParamList));
				stAX5000Diag.bPreopToSafeOpError := FALSE;
				stAX5000Diag.bSafeOpToOpError := FALSE;
				iSubState	:= iSubState + 3;
			END_IF
		END_IF
	
	6:	(* read S21 - IDN List of Invalid operation data for CP2 (Preop->SaveOp) *)
		fbSoERead(
			NetId	:= IPCNetID,
			Execute	:= TRUE,
			Idn		:= 21,
			Element	:=16#40,
			pDstBuf	:=ADR(stAX5000Diag.stCPxInvParamList),
			BufLen	:=SIZEOF(stAX5000Diag.stCPxInvParamList),
			Timeout	:= DEFAULT_ADS_TIMEOUT,
			Axis	:= Axis,
		);
	
		IF NOT fbSoERead.Busy THEN
			fbSoERead(Execute:= FALSE,Axis := Axis);
			IF NOT fbSoERead.Error THEN
				;
			ELSE
				Error			:= TRUE;
				AdsErrId		:= fbSoERead.AdsErrId;
				SercosErrId	:= fbSoERead.SercosErrId;
			END_IF
			iSubState	:= iSubState + 2;
		END_IF
	
	7:	(* read S22 - IDN List of Invalid operation data for CP3 (SaveOp->Op) *)
		fbSoERead(
			NetId	:= IPCNetID,
			Execute	:= TRUE,
			Idn		:= 22,
			Element	:=16#40,
			pDstBuf	:=ADR(stAX5000Diag.stCPxInvParamList),
			BufLen	:=SIZEOF(stAX5000Diag.stCPxInvParamList),
			Timeout	:= DEFAULT_ADS_TIMEOUT,
			Axis	:= Axis,
		);
	
		IF NOT fbSoERead.Busy THEN
			fbSoERead(Execute:= FALSE,Axis := Axis);
			IF NOT fbSoERead.Error THEN
				;
			ELSE
				Error			:= TRUE;
				AdsErrId		:= fbSoERead.AdsErrId;
				SercosErrId	:= fbSoERead.SercosErrId;
			END_IF
			iSubState	:= iSubState + 1;
		END_IF
	
	8:	fbDiagNumberList(
			NetId			:= IPCNetID,
			Execute			:= TRUE,
			Timeout			:= DEFAULT_ADS_TIMEOUT,
			pDiagNumber		:= ADR(stAX5000Diag.stDiagNumberList),
			Size			:= SIZEOF(stAX5000Diag.stDiagNumberList),
			Axis			:= Axis,
		);
	
		IF NOT fbDiagNumberList.Busy THEN
			fbDiagNumberList(Execute:= FALSE,Axis := Axis);

			IF NOT fbDiagNumberList.Error THEN
				IF bLogDriveDiagMsgs THEN
					IF (stAX5000Diag.strDiagMessage <> DiagMsgPrev) AND (stAX5000Diag.stDiagNumberList.iActualSize > 0) THEN
	
						fbFormatString(
							sFormat := 'Axis ID: %d, DriveDiag: ',
							arg1 := F_UDINT(AxisID),
							sOut => LogMsg
						);
		
						FOR I := 0 TO MIN(29, UINT_TO_INT(stAX5000Diag.stDiagNumberList.iActualSize)/4-1) DO
							IF (stAX5000Diag.stDiagNumberList.arrDiagNumbers[I] <> 0) THEN
								fbFormatString(
									sFormat := '%X, ',
									arg1 := F_UDINT(stAX5000Diag.stDiagNumberList.arrDiagNumbers[I])
								);
		
								LogMsg := CONCAT(LogMsg, fbFormatString.sOut);
							END_IF
						END_FOR
		
						LogMsg := CONCAT(LogMsg, 'DiagMsg: ');
						LogMsg := CONCAT(LogMsg, stAX5000Diag.strDiagMessage);
		
						(* report message *)
						ADSLOGSTR(msgCtrlMask := ADSLOG_MSGTYPE_ERROR OR ADSLOG_MSGTYPE_LOG,
							msgFmtStr := LogMsg, strArg:= '');
		
						DiagMsgPrev := stAX5000Diag.strDiagMessage;
					END_IF
				END_IF
			ELSE
				Error			:= TRUE;
				AdsErrId		:= fbDiagNumberList.AdsErrId;
				SercosErrId	:= fbDiagNumberList.SercosErrId;
			END_IF
	
			IF (stAX5000Diag.strMotorType = '') OR (stAX5000Diag.strDriveType = '') THEN
				iSubState	:= iSubState + 1;
			ELSE
				DiagAct	:= FALSE;
				iSubState	:= 0;
				iState		:= 0;
				Busy		:= FALSE;
			END_IF
		END_IF
	
	9:	fbSoERead(
			NetId	:= IPCNetID,
			Execute	:= TRUE,
			Idn		:= P_0_IDN + 53,
			Element	:=16#44,
			pDstBuf	:=ADR(strSoEString),
			BufLen	:=SIZEOF(strSoEString),
			Timeout	:= DEFAULT_ADS_TIMEOUT,
			Axis	:= Axis,
		);
	
		IF NOT fbSoERead.Busy THEN
			fbSoERead(Execute:= FALSE,Axis := Axis);
			IF NOT fbSoERead.Error THEN
				MEMSET(ADR(stAX5000Diag.strMotorType),0,SIZEOF(stAX5000Diag.strMotorType));
				MEMCPY(ADR(stAX5000Diag.strMotorType),ADR(strSoEString.strData),MIN(SIZEOF(stAX5000Diag.strMotorType),strSoEString.iActualSize));
			ELSE
				Error			:= TRUE;
				AdsErrId		:= fbSoERead.AdsErrId;
				SercosErrId	:= fbSoERead.SercosErrId;
			END_IF
			iSubState	:= iSubState + 1;
		END_IF
	
	10:	fbSoERead(
			NetId	:= IPCNetID,
			Execute	:= TRUE,
			Idn		:= P_0_IDN + 324,
			Element	:=16#44,
			pDstBuf	:=ADR(strSoEString),
			BufLen	:=SIZEOF(strSoEString),
			Timeout	:= DEFAULT_ADS_TIMEOUT,
			Axis	:= Axis,
		);
	
		IF NOT fbSoERead.Busy THEN
			fbSoERead(Execute:= FALSE,Axis := Axis);
			IF NOT fbSoERead.Error THEN
				MEMSET(ADR(stAX5000Diag.strDriveType),0,SIZEOF(stAX5000Diag.strDriveType));
				MEMCPY(ADR(stAX5000Diag.strDriveType),ADR(strSoEString.strData),MIN(SIZEOF(stAX5000Diag.strDriveType),strSoEString.iActualSize));
			ELSE
				Error			:= TRUE;
				AdsErrId		:= fbSoERead.AdsErrId;
				SercosErrId	:= fbSoERead.SercosErrId;
			END_IF
			DiagAct	:= FALSE;
			iSubState	:= 0;
			iState		:= 0;
			Busy		:= FALSE;
		END_IF

END_CASE
END_ACTION

ACTION A_GetDriveRef:
(* get reference from NC *)
fbAdsRead(
	NETID	:= IPCNetID,
	PORT	:= AMSPORT_R0_NC,
	IDXGRP	:= NCIDXG_AXPARMS + Axis.NcToPlc.AxisId,
	IDXOFFS	:= NCIDXO_AXP_HWAMSADDR,
	LEN		:= SIZEOF(readBuffer) ,
	DESTADDR:= ADR(readBuffer),
	READ	:= TRUE,
	TMOUT	:= Timeout
);

IF NOT fbAdsRead.BUSY THEN
	fbAdsRead(READ := FALSE);
	stAX5000Diag.nNCAxisID := Axis.NcToPlc.AxisId;

	IF NOT fbAdsRead.ERR THEN
		MEMCPY(ADR(Ids), ADR(readBuffer), SIZEOF(Ids)); 										(* readBuffer[0..5] *)
		MEMCPY(ADR(DriveRef.nSlaveAddr), ADR(readBuffer[6]), SIZEOF(DriveRef.nSlaveAddr));  	(* readBuffer[6..7] *)
		MEMCPY(ADR(DriveRef.nDriveNo), ADR(readBuffer[8]), SIZEOF(DriveRef.nDriveNo));  		(* readBuffer[8..9] *)

		(* create string out of byte array *)
		DriveRef.sNetId := F_CreateAmsNetId(Ids);
		GetDriveRef := FALSE;
	END_IF

	Busy	:= FALSE;
	iState	:= 0;
END_IF
END_ACTION

ACTION A_Reset:

CASE iSubState OF

	0:
		IF stAX5000Diag.bWcStateError OR stAX5000Diag.bC1DError THEN
			(* ResetAmplifier *)
			iSubState := iSubState + 1;
		ELSIF stAX5000Diag.stEcSlaveStateBits.bError AND bForceStateChgAfterDrvReset THEN
			(* Clear Error *)
			iSubState := 4;
		ELSIF (NOT stAX5000Diag.bOperational) OR stAX5000Diag.bAxisError OR (stAX5000Diag.iAxisErrorCode <> 0) THEN
			(* NC Reset only *)
			iSubState := 6;
		ELSE
			(* reset not required *)
			iSubState	:= 0;
			iState		:= 0;
			Busy		:= FALSE;
			ResetAct		:= FALSE;
		END_IF

	1:	(* ResetAmplifier *)
		fbReset(
			NetId	:= IPCNetID,
			Execute	:= TRUE,
			Timeout	:= DEFAULT_ADS_TIMEOUT,
			Axis	:= Axis,
		);
		IF NOT fbReset.Busy THEN
			fbReset(Execute:= FALSE, Axis:= Axis);

			IF NOT fbReset.Error THEN
				IF bLogDriveDiagMsgs THEN
					LogMsg := CONCAT('Axis ID: ', DWORD_TO_STRING(Axis.NcToPlc.AxisId));
					LogMsg := CONCAT(LogMsg, ', Drive Reset');

					(* report message *)
					ADSLOGSTR(msgCtrlMask := ADSLOG_MSGTYPE_ERROR OR ADSLOG_MSGTYPE_LOG,
						msgFmtStr := LogMsg, strArg:= '');

					DiagMsgPrev := '';
				END_IF
				iSubState	:= iSubState + 1;
			ELSE
				Error			:= TRUE;
				AdsErrId		:= fbReset.AdsErrId;
				SercosErrId	:= fbReset.SercosErrId;
				Busy			:= FALSE;
				ResetAct		:= FALSE;
				iSubState		:= 0;
				iState			:= 0;
			END_IF
		END_IF

	2:	fbDelay(IN:=TRUE, PT:=t#3s);
		IF fbDelay.Q THEN
			fbDelay(IN:=FALSE);
			iSubState	:= iSubState + 1;
		END_IF

	3:	fbGetSlaveState(
			sNetId		:= DriveRef.sNetId,
			nSlaveAddr	:= DriveRef.nSlaveAddr,
			bExecute	:= TRUE,
			tTimeout	:= DEFAULT_ADS_TIMEOUT,
		);

		IF NOT fbGetSlaveState.bBusy THEN
			fbGetSlaveState(bExecute:= FALSE);

			IF NOT fbGetSlaveState.bError THEN
		(* Slave in error state	*)
				IF ((fbGetSlaveState.state.deviceState <> 16#08) OR ((fbGetSlaveState.state.deviceState AND 16#10) = 16#10)) AND
					bForceStateChgAfterDrvReset THEN

					iSubState	:= iSubState + 1;
				ELSIF Axis.NcToPlc.StateDWord.31 OR (Axis.NcToPlc.ErrorCode <> 0) THEN
					iSubState	:= 6;
				ELSE
					Busy		:= FALSE;
					ResetAct	:= FALSE;
					iSubState	:= 0;
					iState		:= 0;
					ResetDone := TRUE;
				END_IF
			ELSE
				Error			:= TRUE;
				AdsErrId		:= UDINT_TO_UINT(fbGetSlaveState.nErrId);
				Busy			:= FALSE;
				ResetAct		:= FALSE;
				iSubState		:= 0;
				iState			:= 0;
			END_IF
		END_IF
	
	4:	(* clear error *)
		fbReqSlaveState(
			sNetId		:= DriveRef.sNetId,
			nSlaveAddr	:= DriveRef.nSlaveAddr,
			bExecute	:= TRUE,
			tTimeout	:= DEFAULT_ADS_TIMEOUT,
			state		:= EC_DEVICE_STATE_ERROR);
	
		IF NOT fbReqSlaveState.bBusy THEN
			fbReqSlaveState(bExecute:= FALSE);

			IF NOT fbReqSlaveState.bError THEN
				iSubState	:= iSubState + 1;
			ELSE
				Error		:= TRUE;
				AdsErrId	:= UDINT_TO_UINT(fbReqSlaveState.nErrId);
				Busy		:= FALSE;
				ResetAct	:= FALSE;
				iSubState	:= 0;
				iState		:= 0;
			END_IF
		END_IF
	
	5:	(* set op *)
		fbReqSlaveState(
			sNetId		:= DriveRef.sNetId,
			nSlaveAddr	:= DriveRef.nSlaveAddr,
			bExecute	:= TRUE,
			tTimeout	:= DEFAULT_ADS_TIMEOUT,
			state		:= EC_DEVICE_STATE_OP);

		IF NOT fbReqSlaveState.bBusy THEN
			fbReqSlaveState(bExecute:= FALSE);
	
			IF NOT fbReqSlaveState.bError THEN
				iSubState	:= iSubState + 1;
			ELSE
				Error		:= TRUE;
				AdsErrId	:= UDINT_TO_UINT(fbReqSlaveState.nErrId);
				Busy		:= FALSE;
				ResetAct	:= FALSE;
				iSubState	:= 0;
				iState		:= 0;
			END_IF
		END_IF
	
	6:	fbNcReset(
			Execute:= TRUE,
			Axis:= Axis,
		);
	
		IF fbNcReset.Done OR fbNcReset.Error THEN
			IF fbNcReset.Error THEN
				Error 		:= TRUE;
				AdsErrId 	:= UDINT_TO_UINT(fbNcReset.ErrorID);
			ELSE
				ResetDone := TRUE;
			END_IF
	
			iSubState	:= 0;
			iState		:= 0;
			Busy		:= FALSE;
			ResetAct		:= FALSE;
			fbNcReset(Execute:= FALSE, Axis:= Axis);
		END_IF

END_CASE
END_ACTION

END_FUNCTION_BLOCK

// Motion/Functions/Lenze_84xx/F_DecodeLenze84Status
FUNCTION F_DecodeLenze84Status : ST_84_Status
VAR_INPUT
	InStatusWord			:WORD;
END_VAR
VAR
END_VAR

(* 	Zur SPS vom Regler:
W1 Statuswort New
Bit0		Drive Ready
Bit1		Impulssperre (gesperrt von SPS)
Bit2		free
Bit3		free
Bit4		free
Bit5		free
Bit6		Aktuelle Drehzahl < C24 (Moving..)
Bit7		Reglersperre aktiv
Bit8		ZustandsID Bit 0
Bit9		ZustandsID Bit 1
Bit10 	ZustandsID Bit 2
Bit11 	ZustandsID Bit 3
Bit12 	Warning aktiv
Bit13 	Fail aktiv
Bit14 	free
Bit15 	Motor über Temperatur Grenze	

	über Codierung Bit 8-11
	Drive Operation enabled	(	Bit 8 = 1, Bit 9 = 0, Bit 10 = 1, Bit 11 = 0	)
	QSP aktiv				(	Bit 8 = 1, Bit 9 = 0, Bit 10 = 0, Bit 11 = 1	)
	Drive ready to switch on	(	Bit 8 = 1, Bit 9 = 1, Bit 10 = 0, Bit 11 = 0	)
	-
	- Unterspannung Zwischenkreis -> nicht vorhanden
	- Reglersperre 9400 durch Engineer freizugeben ! -> Reglersperre aktiv


	bDriveReady				:BOOL;	(*	Drive Ready to Move	*)
	bImpulssperre			:BOOL;	(*	Impulssperre (gesperrt von SPS)	*)
	bNotMoving				:BOOL;
	bReglersperreAktiv		:BOOL;
	bDriveReadyToSwitchOn	:BOOL;
	bDriveOperationEnabled	:BOOL;
	bQSPAktiv				:BOOL;
	bWarningAktiv			:BOOL;
	bFailAktiv				:BOOL;
	bMotorTempHigh			:BOOL;
*)

(*	Bit 8 = 1, Bit 9 = 1, Bit 10 = 0, Bit 11 = 0	*)
F_DecodeLenze84Status.bDriveReady := InStatusWord.0;
F_DecodeLenze84Status.bImpulssperre := InStatusWord.1;
F_DecodeLenze84Status.bNotMoving := InStatusWord.6;
F_DecodeLenze84Status.bReglersperreAktiv := InStatusWord.7;
F_DecodeLenze84Status.bDriveReadyToSwitchOn :=InStatusWord.8 AND InStatusWord.9 AND NOT InStatusWord.10 AND NOT InStatusWord.11;
F_DecodeLenze84Status.bDriveOperationEnabled :=InStatusWord.8 AND NOT InStatusWord.9 AND InStatusWord.10 AND NOT InStatusWord.11;
F_DecodeLenze84Status.bQSPAktiv := InStatusWord.8 AND NOT InStatusWord.9 AND NOT InStatusWord.10 AND InStatusWord.11;
F_DecodeLenze84Status.bWarningAktiv := InStatusWord.12;
F_DecodeLenze84Status.bFailAktiv := InStatusWord.13;
F_DecodeLenze84Status.bMotorTempHigh := InStatusWord.15;

END_FUNCTION

// Motion/Lenze_84xx/FB_Antrieb84xxSimple
FUNCTION_BLOCK FB_Antrieb84xxSimple
VAR_IN_OUT
	outArr					: IO_84_Lenze_FW2x ;
	inArr					: IO_84_Lenze_FW2x ;	
END_VAR
VAR_INPUT
	/// component active flag
	bActive				:BOOL;
	/// Gibt an ob ein Fehler autom. quitiert werden soll
	bAutoQuittError		:BOOL := TRUE;
	///Objekt Name
	sName				:STRING;
	///Index des Objekts
	diObjectIndex		:DINT;
	/// Sicherheit = Freigabe von Bewegungen
	bSafetyOk			:BOOL;
	/// Hardware OK
	bPowerSupplyOk		:BOOL;
	
	// Hand
	///Ausgewähltes Objekt in der Visu
	diSelectedObjectIndex	:DINT;
	/// Gibt den Handbetrieb frei
	bEnableManual: BOOL;
	// Handbetrieb nach Positiv
	bManual_Pos: BOOL;
	/// Handbetrieb nach Negativ
	bManual_Neg: BOOL;

	// Spezifische Variablen
	fVeloSoll			:REAL := 0;		(*	mm/sek	*)
	fTourqeSoll			:REAL := 100;	(* [100] % -> Drehmomentsollwert in Prozent	*)
	eDirection			:E_DIRECTION;
	bStart				:BOOL;
	bSetPos0			:BOOL;			(*	Aktuelle Position auf 0 setzen	*)
	TipVel				:REAL := 1.0 ;	(* [1.0] mm/sek langsame tipgeschwindigkeit *)

	bTipFast			:BOOL;			(*	schnelles Tippen mit UpmTipFakt	*)
	UpmTipFakt			:REAL := 10;	(* [10] Vervielfachung Drehzahl bei Tippen *)
	
	(*	Einstellungen	*)
	b_RevMot		: BOOL := FALSE ;		(* Motordrehrichtung umkehren *)
	b_RevCount		: BOOL := FALSE;		(* Zählrichtung umkehren *)
	PosFakt			: REAL := 0.001;	(* 	[0.000152587890625] = 10mm Spindel / 2^16 (Steps/Umdr.)
	 										[0.0000762939453125] = 5mm Spindel / 2^16 (Steps/Umdr.)
											[0.0000152587890625] = 1 U / 2^16 (Steps/Umdr.)		*)
	TipRamp		: REAL := 1 ;			(* [1] Rampe pro sekunde *)
	(* Parameter zum Positionieren *)
	UpmMax			: REAL := 1000;			(* [1000] Maximale Drehzahl entsprechend Motor *)
	UpmPsec 		: REAL := 40000 ;			(* [5000] Rampe Upm/sek *)
	bRFR			: BOOL := TRUE ;

	bBremseLoesen		:BOOL;
	bIgnoreError		:BOOL;	
END_VAR
VAR_OUTPUT	
	/// Fehler
	bError				:BOOL;
	/// Fehlertext
	sErrText			:STRING;
	///Darstellung der Controls für das Object 
	///0=Unsichtbar
	///1=Sichtbar Unselektiert
	///2=Sichtbar Selektiert	
	iVisibleState: INT;
	/// 0=Undefiniert
	/// 1=Fehler
	/// 2=In GRST (eingefahren)
	/// 3=In AST (ausgefahren) 
	iStatus: INT;
	
	Qmoving			: BOOL;		(*	Antrieb bewegt sich	*)

	UpmIst			: REAL;		(* [upm] Drehzahl Istwert *)
	MomIst			: REAL;		(* [%] des Nennmmentes Drehmoment istwert *)
	PosIst			: REAL;		(* [mm] Aktuelle Position	*)
	
	/// Aktuelle Positionen mit gelatchten Objektposition gleich
	bLatchedObjPositionOK					:BOOL;
END_VAR
VAR
	LenzeOut  				: ST_84_PLC_to_Lenze ;	(*Strukturausgangsbits*)
	LenzeIn 				: ST_84_Lenze_to_PLC;	(*Struktureingangsbits*)
	strct_LenzeStatus		: ST_84_Status;

	I_Pos_x			: DINT ;				(* zum Vergleich für Überträge *)

	IncTipRamp 		: REAL ;
	di_Zkorr 			: DINT;				(* aktuelle Korrektur mit Nullung etc. *)
	UpmTip			: REAL ;				(* Drehzahl bei Tippen berechnet aus TipVel *)
	UpmVel			: REAL ;				(* Upm berechnet aus = mm/sek * 60 / PosFakt *)
	UpmFakt			: REAL := 16.384;		(* [16.384] = 2^14 / 1000 upm Nenndrehzahl *)
	MomFakt		: REAL := 163.84;		(* [163.84] = 2^14 / 100 %  *)
	UpmSoll			: REAL;
	UpmInc 			: REAL ;				(* Berechnetes Incremet für Rampe *)
	UpmRmp		: REAL;
	UpmOut			: REAL ;	(*	Ausgabe	Drehzahl		*)

	tError			: TON;
	ttError			: TIME := t#1000ms;
	ErrorQuit		: BOOL;					(* Toggelt bei Error zum Reset *)

	bTipAny			:BOOL;
	tTip				: TON;
	ttTip			: TIME := t#500ms;

	b_TestIO			:BOOL;
	b_StartLokal		:BOOL := FALSE ;		(* für Test und Reparatur, Bedienung über TC_Visu *)

	bInit			:BOOL;
END_VAR
VAR PERSISTENT
	PosRoh		:REAL;
	fPosLatched	:REAL;
END_VAR

(*
	Ansteuerung von Motoren ueber Lenze 84er EtherCAT
	TwinCAT 3
	2011-2015 / www.rmth.at / RE
	
*************************************************************************)

// nicht aktiv -> alles löschen und Exit
IF NOT bActive THEN
	bError := FALSE ;
	sErrText := '';
	iStatus := 0;/// 0=Undefiniert
	iVisibleState := 0;
	bStart := FALSE;
	UpmOut := 0;
	RETURN;
END_IF

// Objekt ausgewaehlt
IF (diObjectIndex = diSelectedObjectIndex) THEN
	iVisibleState := 2;	// 2=Sichtbar Selektiert
ELSE
	iVisibleState := 1;	// 1=Sichtbar Unselektiert
END_IF

//
// Lenze Logik
//

(* Lenze Output Daten an PLC Struktur  mit Hilfe einer Überlagerung übergeben *)
MEMCPY(ADR(LenzeIn), ADR(InArr), SIZEOF(LenzeIn));
strct_LenzeStatus := F_DecodeLenze84Status(LenzeIn.wStatus);

(*	wenn Test dann keine IO Belegung durch Baustein	*)
IF b_TestIO THEN
	A_Test( );
	MEMCPY(ADR(outArr), ADR(LenzeOut), SIZEOF(LenzeOut));
	RETURN;	(*	Exit aus FB -> keine Logik	*)
END_IF

A_Error( );

(* Rampen-Werte immer berechnen damit online-Change möglich *)
IncTipRamp := TipRamp * Statics.stPlcSystemInfo.fCycleTime * 1E-7 ;
UpmFakt := 16384 / UpmMax;	(* [16.384] = 2^14 / 1000 upm Nenndrehzahl *)
MomFakt := 16384 / 100;		(* [163.84] = 2^14 / 100 %  *)

UpmIst := LenzeIn.nIstDrz / UpmFakt ;
MomIst := LenzeIn.nIstMom  / MomFakt ;

IF NOT bInit THEN

	IF LenzeIn.nResolverPos = 0 AND LenzeIn.wStatus = 0 THEN
		RETURN;
	ELSE
		bInit := TRUE;
	END_IF

	(*	Restore saved Persistent Pos	*)
	IF b_RevCount THEN
		di_Zkorr := - LenzeIn.nResolverPos - REAL_TO_DINT( PosRoh / PosFakt );
	ELSE
		di_Zkorr := - LenzeIn.nResolverPos + REAL_TO_DINT( PosRoh / PosFakt );
	END_IF
END_IF

UpmTip := LIMIT( 0, TipVel / (PosFakt * 65536) * 60 ,  UpmMax ) ;	(* Umrechnung mm/sek --> upm *)
UpmVel := UpmMax  ;	(* Maximalgeschwindigkeit *)
 (* Rampen-Werte immer berechnen damit online-Change möglich *)
upmInc := UpmPsec * Statics.stPlcSystemInfo.fCycleTime * 1E-7 ;

(*	Tippen	*)
bTipAny := 	(bEnableManual AND bManual_Pos AND (diObjectIndex = diSelectedObjectIndex)) OR
		 	(bEnableManual AND bManual_Neg AND (diObjectIndex = diSelectedObjectIndex)) AND
			bSafetyOk AND bPowerSupplyOk;

tTip(in := bTipAny , pt := ttTip ) ;

// Sicherheit
IF NOT bSafetyOk THEN
	UpmSoll := 0;

// Versorgung NOK 
ELSIF NOT bPowerSupplyOk THEN
	UpmSoll := 0;

ELSIF bStart OR b_StartLokal THEN
	IF eDirection = FORWARD THEN
		UpmSoll := fVeloSoll / (PosFakt * 65536) * 60;	(* Umrechnung mm/sek --> upm *)
	ELSIF eDirection = BACKWARD THEN
		UpmSoll := - fVeloSoll / (PosFakt * 65536) * 60;	(* Umrechnung mm/sek --> upm *)
	ELSE
		UpmSoll := 0;
	END_IF
ELSE
	IF tTip.Q THEN
		IF bManual_Pos THEN (* langsam/schnell + *)
			UpmSoll := TipVel / (PosFakt * 65536) * 60;	(* Umrechnung mm/sek --> upm *) ;
		ELSIF bManual_Neg THEN (* langsam/schnell - *)
			UpmSoll := - TipVel / (PosFakt * 65536) * 60;	(* Umrechnung mm/sek --> upm *) ; ;
		ELSE
			UpmSoll := 0;
		END_IF
		IF bTipFast THEN
			UpmSoll := UpmSoll * UpmTipFakt ;
		END_IF
	ELSE
		UpmSoll := 0;
	END_IF
END_IF

(*	Soll begrenzen	*)
UpmSoll := LIMIT(-UpmMax ,UpmSoll, UpmMax);

A_CalcPosition( );

(*	Bremsen / Beschleunigen	*)
IF UpmRmp > UpmSoll THEN (* Bremsen mit Rampe *)
	UpmRmp := MAX( ( UpmRmp - UpmInc  ) , UpmSoll );
ELSE	(* Beschleunigen mit Rampe *)
	UpmRmp := MIN( ( UpmRmp + UpmInc  ) , UpmSoll );
END_IF

(*	Ausgabe an Antrieb	*)
UpmOut := LIMIT( - UpmVel, UpmRmp , UpmVel ) ;

// Sicherheit
IF NOT bSafetyOk THEN
	UpmOut := 0 ;
	UpmRmp := 0 ;
	LenzeOut.nSollDrz   := 0 ;
	LenzeOut.wControl := 16#0 ;
	LenzeOut.wControl.7 := ErrorQuit ;
	LenzeOut.wControl.8 := bBremseLoesen ;

// Versorgung NOK 
ELSIF NOT bPowerSupplyOk THEN
	UpmOut := 0 ;
	UpmRmp := 0 ;
	LenzeOut.nSollDrz   := 0 ;
	LenzeOut.wControl := 16#0 ;
	LenzeOut.wControl.7 := ErrorQuit ;
	LenzeOut.wControl.8 := bBremseLoesen ;

ELSIF bError THEN
	UpmOut := 0 ;
	UpmRmp := 0 ;
	LenzeOut.nSollDrz   := 0 ;
	LenzeOut.wControl := 16#0 ;
	LenzeOut.wControl.7 := ErrorQuit ;
	LenzeOut.wControl.8 := bBremseLoesen ;

ELSIF bStart OR bTipAny OR b_StartLokal THEN
	LenzeOut.wControl.0 := TRUE ;
	LenzeOut.wControl.3 := bRFR ;	(* RFR wird normalerweise im 84xx von Bremsenmodul abgeschaltet *)
	LenzeOut.wControl.7 := FALSE ;
	LenzeOut.wControl.8 := bBremseLoesen   ;
	IF b_RevMot THEN
		LenzeOut.nSollDrz  := - REAL_TO_INT(LIMIT(-32767.0, (UpmOut * UpmFakt), 32767));
	ELSE
		LenzeOut.nSollDrz  :=   REAL_TO_INT(LIMIT(-32767.0, (UpmOut * UpmFakt), 32767));
	END_IF
ELSE
	LenzeOut.wControl.0 := FALSE;
	LenzeOut.wControl.7 := FALSE ;
	LenzeOut.wControl.8 := bBremseLoesen   ;
	LenzeOut.nSollDrz := 0;
END_IF

LenzeOut.nMaxMom := REAL_TO_INT(LIMIT(-32767.0, (fTourqeSoll * MomFakt), 32767));

Qmoving := LenzeOut.nSollDrz <> 0 AND strct_LenzeStatus.bDriveReady;

(*  PLC Struktur an Lenze Input Daten  mit Hilfe einer Überlagerung übergeben *)
MEMCPY(ADR(outArr), ADR(LenzeOut), SIZEOF(LenzeOut));

// check Latched state
A_CheckLatchState();

ACTION A_CalcPosition:
(*	Position auf 0 setzen	*)
IF bSetPos0 THEN
	di_Zkorr :=  - LenzeIn.nResolverPos ;
	bSetPos0 := FALSE;
END_IF

(*	Position berechnen	*)
IF b_RevCount THEN
	PosRoh := - DINT_TO_REAL(LenzeIn.nResolverPos + di_Zkorr) * PosFakt;
ELSE
	PosRoh := DINT_TO_REAL(LenzeIn.nResolverPos + di_Zkorr) * PosFakt;
END_IF

PosIst := PosRoh;
END_ACTION

ACTION A_CheckLatchState:
bLatchedObjPositionOK := ABS(PosIst - fPosLatched) <= 0.1;
END_ACTION

ACTION A_Error:

(* Fehlerzustand des Lenze 94xx Reglers bearbeiten *)
bError := 	strct_LenzeStatus.bFailAktiv			(* Fehler *)
		OR (NOT strct_LenzeStatus.bDriveReadyToSwitchOn AND	(*	nicht einschaltbereit	*)
			NOT strct_LenzeStatus.bDriveReady); 	(* nicht Ready *)
IF bIgnoreError THEN
	bError := FALSE;
END_IF

(*	Fehlertext	*)
IF bError THEN
	IF strct_LenzeStatus.bFailAktiv THEN
		sErrText := 'Umrichter Fehler aktiv';
	ELSIF NOT strct_LenzeStatus.bDriveReadyToSwitchOn THEN
		sErrText := 'Umrichter nicht einschaltbereit';
	ELSIF NOT strct_LenzeStatus.bDriveReady THEN
		sErrText := 'Umrichter nicht bereit';
	END_IF

ELSE
	sErrText := '';
END_IF

tError( in := bError AND NOT tError.Q , pt := ttError ) ;
IF tError.Q AND bAutoQuittError THEN
	ErrorQuit := NOT ErrorQuit ;
END_IF
IF NOT bError THEN
	ErrorQuit := FALSE ;
END_IF
END_ACTION

ACTION A_Test:
(*	Test		*)
(*
LenzeOut.wControl.0;	(*	Drive Switched On (ON nach Sperre)	*)
LenzeOut.wControl.1;	(*	Impulssperre 	*)
LenzeOut.wControl.2;	(*	QSP	*)
LenzeOut.wControl.3;	(*	RFR	*)
LenzeOut.wControl.4;	(*		*)
LenzeOut.wControl.5;	(*		*)
LenzeOut.wControl.6;	(*		*)
LenzeOut.wControl.7;	(*	Trip Reset	*)
LenzeOut.wControl.8;	(*	Break release	*)
LenzeOut.wControl.9;	(*		*)
LenzeOut.wControl.10;	(*		*)
LenzeOut.wControl.11;	(*		*)
LenzeOut.wControl.12;	(*	Jog 1	*)
LenzeOut.wControl.13;	(*		*)
LenzeOut.wControl.14;	(*		*)
LenzeOut.wControl.15;	(*	Drehrichtungsumkehr*)

LenzeOut.nSollDrz;

LenzeIn.wStatus.0;		(*	Drive Ready	*)
LenzeIn.wStatus.1;		(*	Impulssperre (gesperrt von SPS)		*)
LenzeIn.wStatus.2;		(*		*)
LenzeIn.wStatus.3;		(*		*)
LenzeIn.wStatus.4;		(*		*)
LenzeIn.wStatus.5;		(*		*)
LenzeIn.wStatus.6;		(*	Aktuelle Drehzahl < C24 (Moving..)	*)
LenzeIn.wStatus.7;		(*	Reglersperre aktiv		*)
LenzeIn.wStatus.8;		(*	ZustandsID Bit 0	*)
LenzeIn.wStatus.9;		(*	ZustandsID Bit 1	*)
LenzeIn.wStatus.10;	(*	ZustandsID Bit 2	*)
LenzeIn.wStatus.11;	(*	ZustandsID Bit 3	*)
LenzeIn.wStatus.12;	(*	Warning aktiv		*)
LenzeIn.wStatus.13;	(*	Fail aktiv		*)
LenzeIn.wStatus.14;	(*		*)
LenzeIn.wStatus.15;	(*	Motor über Temperatur Grenze		*)
*)
END_ACTION

/// Methode um Status des Objekt zu speichern
METHOD LatchObjState : BOOL
fPosLatched := PosIst;
END_METHOD

METHOD Reset
VAR
END_VAR
END_METHOD

END_FUNCTION_BLOCK

// Motion/LenzeIndraDiag/FB_IndraDriveDiag
FUNCTION_BLOCK FB_IndraDriveDiag
VAR_INPUT
	sIPCNetID			: T_AmsNetId; 	(* AmsNetId of the IPC *)
	tTimeout			: TIME := DEFAULT_ADS_TIMEOUT;
	bReset				: BOOL;
	bGetDiag			: BOOL;
END_VAR
VAR_IN_OUT
	Axis				: AXIS_REF;
	stDriveDiag			: ST_IndraDriveDiag;
END_VAR
VAR_OUTPUT
	bError				: BOOL;
	iAdsErrId			: UINT;
	iSercosErrId		: UINT;
	bResetAct			: BOOL;
	bDiagAct			: BOOL;
	bBusy				: BOOL;
END_VAR
VAR
	iState				: INT;
	iSubState			: INT;
	bGetDriveRef		: BOOL := TRUE;
	stDriveRef			: ST_DriveRef; (* contains sNetID of EcMaster, nSlaveAddr of EcDrive, nDriveNo of EcDrive, either preset or read from NC *)
	iAxisID				: UDINT;

	bC1DErrorPrev		: BOOL;
	bWcStateErrorPrev	: BOOL;
	bAxisErrorPrev		: BOOL;
	bOperationalPrev	: BOOL;
	bResetPrev			: BOOL;
	bGetDiagPrev		: BOOL;

	fbSoERead			: FB_SoERead;
	fbDiagMessage 		: FB_SoEReadDiagMessage;
	fbClassXDiag		: FB_SoEReadClassXDiag;
	fbDiagNumber		: FB_SoEReadDiagNumber;
	fbDiagNumberList	: FB_SoEReadDiagNumberList;

	fbReset				: FB_SoEReset;
	fbDelay				: TON;
	fbGetSlaveState 	: FB_EcGetSlaveState;
	fbReqSlaveState 	: FB_EcReqSlaveState;
	fbNcReset 			: MC_Reset;

	fbAdsRead			: ADSREAD;
	readBuffer			: ARRAY[0..9] OF BYTE;
	nIds				: T_AmsNetIdArr;

	fbFormatString		: FB_FormatString;
	strDiagMsgPrev		: STRING(255);
	strLogMsg			: STRING(255);
	strSoEString		: ST_SoE_StringEx;
	I					: INT;
END_VAR
VAR CONSTANT
	NCIDXG_AXPARMS			: UDINT := 16#00004000;	(* Axis with ID: Parameter 			*)
	NCIDXO_AXP_HWAMSADDR	: UDINT := 16#00000031;
END_VAR

stDriveDiag.bOperational	:= Axis.NcToPlc.StateDWord.0;
stDriveDiag.bC1DError	 	:= Axis.NcToPlc.StateDWord.28;
stDriveDiag.bWcStateError 	:= Axis.NcToPlc.StateDWord.30;
stDriveDiag.bAxisError		:= Axis.NcToPlc.StateDWord.31;
stDriveDiag.iAxisErrorCode	:= Axis.NcToPlc.ErrorCode;

CASE iState OF
0:	(* idle *)
	bGetDriveRef 	:= (stDriveRef.nSlaveAddr = 0);

	IF bGetDriveRef THEN
		bBusy			:= TRUE;
		bError			:= FALSE;
		iAdsErrId		:= 0;
		iSercosErrId	:= 0;
		iState 			:= 1;
		iSubState		:= 0;
		iAxisID 		:= Axis.NcToPlc.AxisId;

	ELSIF bReset AND NOT bResetPrev THEN
		bBusy			:= TRUE;
		bResetAct		:= TRUE;
		bResetPrev		:= bReset;
		bError			:= FALSE;
		iAdsErrId		:= 0;
		iSercosErrId	:= 0;
		iState 			:= 2;
		iSubState		:= 0;
		iAxisID 		:= Axis.NcToPlc.AxisId;

	ELSIF bGetDiag AND NOT bGetDiagPrev OR
		(stDriveDiag.bC1DError AND NOT bC1DErrorPrev) OR (NOT stDriveDiag.bC1DError AND bC1DErrorPrev) (* rising/falling C1D *) OR
		(stDriveDiag.bWcStateError AND NOT bWcStateErrorPrev) OR (NOT stDriveDiag.bWcStateError AND bWcStateErrorPrev) (* rising/falling WcState *) OR
		(stDriveDiag.bAxisError AND NOT bAxisErrorPrev) OR (NOT stDriveDiag.bAxisError AND bAxisErrorPrev) (* rising/falling NcError *) OR
		(stDriveDiag.bOperational AND NOT bOperationalPrev) OR (NOT stDriveDiag.bOperational AND bOperationalPrev) (* rising/falling Enable *) THEN

		bBusy			:= TRUE;
		bDiagAct		:= TRUE;
		bGetDiagPrev	:= bGetDiag;
		bError			:= FALSE;
		iAdsErrId		:= 0;
		iSercosErrId	:= 0;
		iState 			:= 3;
		iSubState		:= 0;
		iAxisID 		:= Axis.NcToPlc.AxisId;

		(* set/clear flags *)
		bC1DErrorPrev		:= stDriveDiag.bC1DError;
		bWcStateErrorPrev	:= stDriveDiag.bWcStateError;
		bAxisErrorPrev		:= stDriveDiag.bAxisError;
		bOperationalPrev	:= stDriveDiag.bOperational;

	ELSE
		bResetAct		:= FALSE;
		bDiagAct		:= FALSE;
	END_IF

1:	(* get drive reference *)
	A_GetDriveRef();

2:	(* reset and state change *)
	A_Reset();

3:	(* get diag data *)
	A_GetDiagnosis();

END_CASE

(* clear latch *)
bResetPrev		:= bResetPrev AND bReset;
bGetDiagPrev	:= bGetDiagPrev AND bGetDiag;

ACTION A_GetDiagnosis:
CASE iSubState OF
0:	fbClassXDiag(
		NetId		:= sIPCNetID,
		Execute	:= TRUE,
		DiagClass 	:= 1,
		Timeout	:= DEFAULT_ADS_TIMEOUT,
		Axis		:= Axis,
	);

	IF NOT fbClassXDiag.Busy THEN
		fbClassXDiag(Execute:= FALSE,Axis := Axis);

		IF NOT fbClassXDiag.Error THEN
			stDriveDiag.wClass1Diag		:= fbClassXDiag.ClassXDiag;
			stDriveDiag.stClass1Diag	:= F_ConvWordToSTIndraDriveCsC1D(stDriveDiag.wClass1Diag);
		ELSE
			bError			:= TRUE;
			iAdsErrId		:= fbClassXDiag.AdsErrId;
			iSercosErrId	:= fbClassXDiag.SercosErrId;
		END_IF
		iSubState	:= iSubState + 1;
	END_IF

1:	fbDiagMessage(
		NetId	:= sIPCNetID,
		Execute:= TRUE,
		Timeout:= DEFAULT_ADS_TIMEOUT,
		Axis	:= Axis,
	);

	IF NOT fbDiagMessage.Busy THEN
		fbDiagMessage(Execute:= FALSE,Axis := Axis);

		IF NOT fbDiagMessage.Error THEN
			stDriveDiag.strDiagMessage := LEFT(fbDiagMessage.DiagMessage.strData, fbDiagMessage.DiagMessage.iActualSize);
		ELSE
			bError			:= TRUE;
			iAdsErrId		:= fbDiagMessage.AdsErrId;
			iSercosErrId	:= fbDiagMessage.SercosErrId;
		END_IF
		iSubState	:= iSubState + 1;
	END_IF

2:	fbDiagNumber(
		NetId	:= sIPCNetID,
		Execute:= TRUE,
		Timeout:= DEFAULT_ADS_TIMEOUT,
		Axis	:= Axis,
	);

	IF NOT fbDiagNumber.Busy THEN
		fbDiagNumber(Execute:= FALSE,Axis := Axis);

		IF NOT fbDiagNumber.Error THEN
			stDriveDiag.iDiagNumber := fbDiagNumber.DiagNumber;
		ELSE
			bError			:= TRUE;
			iAdsErrId		:= fbDiagNumber.AdsErrId;
			iSercosErrId	:= fbDiagNumber.SercosErrId;
		END_IF
		iSubState	:= iSubState + 1;
	END_IF

3:	fbSoERead(
		NetId	:= sIPCNetID,
		Execute:= TRUE,
		Idn	:= 135,
		Element:=16#44, (* EC_SOE_ELEMENT_VALUE | EC_SOE_ELEMENT_ATTRIBUTE *)
		pDstBuf	:=ADR(stDriveDiag.wDriveStatus),
		BufLen:=SIZEOF(stDriveDiag.wDriveStatus),
		Timeout:= DEFAULT_ADS_TIMEOUT,
		Axis	:= Axis,
	);

	IF NOT fbSoERead.Busy THEN
		fbSoERead(Execute:= FALSE,Axis := Axis);
		IF NOT fbSoERead.Error THEN
			stDriveDiag.stDriveStatus := F_ConvWordToSTIndraDriveCsDriveStatus(stDriveDiag.wDriveStatus);
			iSubState		:= iSubState + 1;
		ELSE
			bError			:= TRUE;
			iAdsErrId		:= fbSoERead.AdsErrId;
			iSercosErrId	:= fbSoERead.SercosErrId;
			iSubState		:= iSubState + 2;
		END_IF
	END_IF

4:	fbSoERead(
		NetId	:= sIPCNetID,
		Execute:= TRUE,
		Idn	:= stDriveDiag.stDriveStatus.iActOpModeParNum,
		Element:=16#44, (* EC_SOE_ELEMENT_VALUE | EC_SOE_ELEMENT_ATTRIBUTE *)
		pDstBuf	:=ADR(stDriveDiag.stDriveStatus.eActOpMode),
		BufLen:=SIZEOF(stDriveDiag.stDriveStatus.eActOpMode),
		Timeout:= DEFAULT_ADS_TIMEOUT,
		Axis	:= Axis,
	);

	IF NOT fbSoERead.Busy THEN
		fbSoERead(Execute:= FALSE,Axis := Axis);
		IF NOT fbSoERead.Error THEN
			;
		ELSE
			bError			:= TRUE;
			iAdsErrId		:= fbSoERead.AdsErrId;
			iSercosErrId	:= fbSoERead.SercosErrId;
		END_IF
		iSubState	:= iSubState + 1;
	END_IF

5:	fbGetSlaveState(
		sNetId		:= stDriveRef.sNetId,
		nSlaveAddr	:= stDriveRef.nSlaveAddr,
		bExecute	:= TRUE,
		tTimeout	:= DEFAULT_ADS_TIMEOUT,
	);

	IF NOT fbGetSlaveState.bBusy THEN
		fbGetSlaveState(bExecute:= FALSE);
		IF NOT fbGetSlaveState.bError THEN
			stDriveDiag.stEcSlaveState := fbGetSlaveState.state;
			stDriveDiag.stEcSlaveStateBits := F_ConvSlaveStateToBits(fbGetSlaveState.state);
		ELSE
			bError			:= TRUE;
			iAdsErrId		:= UDINT_TO_UINT(fbGetSlaveState.nErrId);
		END_IF

		IF stDriveDiag.stEcSlaveStateBits.bError THEN
			IF stDriveDiag.stEcSlaveStateBits.bPreop THEN
				(* read S21 - IDN List of Invalid operation data for CP2 (Preop->SaveOp) *)
				MEMSET(ADR(stDriveDiag.stCPxInvParamList), 0, SIZEOF(stDriveDiag.stCPxInvParamList));
				stDriveDiag.bPreopToSafeOpError := TRUE;
				stDriveDiag.bSafeOpToOpError := FALSE;
				iSubState	:= iSubState + 1;
			ELSIF stDriveDiag.stEcSlaveStateBits.bSafeOp THEN
				(* read S22 - IDN List of Invalid operation data for CP3 (SaveOp->Op) *)
				MEMSET(ADR(stDriveDiag.stCPxInvParamList), 0, SIZEOF(stDriveDiag.stCPxInvParamList));
				stDriveDiag.bPreopToSafeOpError := FALSE;
				stDriveDiag.bSafeOpToOpError := TRUE;
				iSubState	:= iSubState + 2;
			ELSE
				(* Skip S21 + S22 *)
				MEMSET(ADR(stDriveDiag.stCPxInvParamList), 0, SIZEOF(stDriveDiag.stCPxInvParamList));
				stDriveDiag.bPreopToSafeOpError := FALSE;
				stDriveDiag.bSafeOpToOpError := FALSE;
				iSubState	:= iSubState + 3;
			END_IF
		ELSE
			(* Skip S21 + S22 *)
			MEMSET(ADR(stDriveDiag.stCPxInvParamList), 0, SIZEOF(stDriveDiag.stCPxInvParamList));
			stDriveDiag.bPreopToSafeOpError := FALSE;
			stDriveDiag.bSafeOpToOpError := FALSE;
			iSubState	:= iSubState + 3;
		END_IF
	END_IF

6:	(* read S21 - IDN List of Invalid operation data for CP2 (Preop->SaveOp) *)
	fbSoERead(
		NetId	:= sIPCNetID,
		Execute:= TRUE,
		Idn	:= 21,
		Element:=16#40, (* EC_SOE_ELEMENT_VALUE *)
		pDstBuf	:=ADR(stDriveDiag.stCPxInvParamList),
		BufLen:=SIZEOF(stDriveDiag.stCPxInvParamList),
		Timeout:= DEFAULT_ADS_TIMEOUT,
		Axis	:= Axis,
	);

	IF NOT fbSoERead.Busy THEN
		fbSoERead(Execute:= FALSE,Axis := Axis);
		IF NOT fbSoERead.Error THEN
			;
		ELSE
			bError			:= TRUE;
			iAdsErrId		:= fbSoERead.AdsErrId;
			iSercosErrId	:= fbSoERead.SercosErrId;
		END_IF
		iSubState	:= iSubState + 2;
	END_IF

7:	(* read S22 - IDN List of Invalid operation data for CP3 (SaveOp->Op) *)
	fbSoERead(
		NetId	:= sIPCNetID,
		Execute:= TRUE,
		Idn	:= 22,
		Element:=16#40, (* EC_SOE_ELEMENT_VALUE *)
		pDstBuf	:=ADR(stDriveDiag.stCPxInvParamList),
		BufLen:=SIZEOF(stDriveDiag.stCPxInvParamList),
		Timeout:= DEFAULT_ADS_TIMEOUT,
		Axis	:= Axis,
	);

	IF NOT fbSoERead.Busy THEN
		fbSoERead(Execute:= FALSE,Axis := Axis);
		IF NOT fbSoERead.Error THEN
			;
		ELSE
			bError			:= TRUE;
			iAdsErrId		:= fbSoERead.AdsErrId;
			iSercosErrId	:= fbSoERead.SercosErrId;
		END_IF
		iSubState	:= iSubState + 1;
	END_IF

8:	fbDiagNumberList(
		NetId			:= sIPCNetID,
		Execute		:= TRUE,
		Timeout		:= DEFAULT_ADS_TIMEOUT,
		pDiagNumber	:= ADR(stDriveDiag.stDiagNumberList),
		Size			:= SIZEOF(stDriveDiag.stDiagNumberList),
		Axis			:= Axis,
	);

	IF NOT fbDiagNumberList.Busy THEN
		fbDiagNumberList(Execute:= FALSE,Axis := Axis);

		IF NOT fbDiagNumberList.Error THEN
			IF bLogDriveDiagMsgs THEN
				IF (stDriveDiag.strDiagMessage <> strDiagMsgPrev) AND (stDriveDiag.stDiagNumberList.iActualSize > 0) THEN

					fbFormatString(
						sFormat := 'Axis ID: %d, DriveDiag: ',
						arg1 := F_UDINT(iAxisID),
						sOut => strLogMsg
					);

					FOR I := 0 TO MIN(49, stDriveDiag.stDiagNumberList.iActualSize/4-1) DO
						IF (stDriveDiag.stDiagNumberList.arrDiagNumbers[I] <> 0) THEN
							fbFormatString(
								sFormat := '%X, ',
								arg1 := F_UDINT(stDriveDiag.stDiagNumberList.arrDiagNumbers[I])
							);
	
							strLogMsg := CONCAT(strLogMsg, fbFormatString.sOut);
						END_IF
					END_FOR
	
					strLogMsg := CONCAT(strLogMsg, 'DiagMsg: ');
					strLogMsg := CONCAT(strLogMsg, stDriveDiag.strDiagMessage);
	
					(* report message *)
					ADSLOGSTR(msgCtrlMask := ADSLOG_MSGTYPE_ERROR OR ADSLOG_MSGTYPE_LOG,
						msgFmtStr := strLogMsg, strArg:= '');
	
					strDiagMsgPrev := stDriveDiag.strDiagMessage;
				END_IF
			END_IF
		ELSE
			bError			:= TRUE;
			iAdsErrId		:= fbDiagNumberList.AdsErrId;
			iSercosErrId	:= fbDiagNumberList.SercosErrId;
		END_IF

		IF (stDriveDiag.strMotorType = '') OR (stDriveDiag.strDriveType = '') THEN
			iSubState	:= iSubState + 1;
		ELSE
			bDiagAct	:= FALSE;
			iSubState	:= 0;
			iState		:= 0;
			bBusy		:= FALSE;
		END_IF
	END_IF

9:	fbSoERead(
		NetId	:= sIPCNetID,
		Execute:= TRUE,
		Idn	:= S_0_IDN + 141,
		Element:=16#44, (* EC_SOE_ELEMENT_VALUE | EC_SOE_ELEMENT_ATTRIBUTE *)
		pDstBuf	:=ADR(strSoEString),
		BufLen:=SIZEOF(strSoEString),
		Timeout:= DEFAULT_ADS_TIMEOUT,
		Axis	:= Axis,
	);

	IF NOT fbSoERead.Busy THEN
		fbSoERead(Execute:= FALSE,Axis := Axis);
		IF NOT fbSoERead.Error THEN
			MEMSET(ADR(stDriveDiag.strMotorType),0,SIZEOF(stDriveDiag.strMotorType));
			MEMCPY(ADR(stDriveDiag.strMotorType),ADR(strSoEString.strData),MIN(SIZEOF(stDriveDiag.strMotorType),strSoEString.iActualSize));
		ELSE
			bError			:= TRUE;
			iAdsErrId		:= fbSoERead.AdsErrId;
			iSercosErrId	:= fbSoERead.SercosErrId;
		END_IF
		iSubState	:= iSubState + 1;
	END_IF

10:	fbSoERead(
		NetId	:= sIPCNetID,
		Execute:= TRUE,
		Idn	:= S_0_IDN + 140,
		Element:=16#44, (* EC_SOE_ELEMENT_VALUE | EC_SOE_ELEMENT_ATTRIBUTE *)
		pDstBuf	:=ADR(strSoEString),
		BufLen:=SIZEOF(strSoEString),
		Timeout:= DEFAULT_ADS_TIMEOUT,
		Axis	:= Axis,
	);

	IF NOT fbSoERead.Busy THEN
		fbSoERead(Execute:= FALSE,Axis := Axis);
		IF NOT fbSoERead.Error THEN
			MEMSET(ADR(stDriveDiag.strDriveType),0,SIZEOF(stDriveDiag.strDriveType));
			MEMCPY(ADR(stDriveDiag.strDriveType),ADR(strSoEString.strData),MIN(SIZEOF(stDriveDiag.strDriveType),strSoEString.iActualSize));
		ELSE
			bError			:= TRUE;
			iAdsErrId		:= fbSoERead.AdsErrId;
			iSercosErrId	:= fbSoERead.SercosErrId;
		END_IF
		bDiagAct	:= FALSE;
		iSubState	:= 0;
		iState		:= 0;
		bBusy		:= FALSE;
	END_IF


END_CASE
END_ACTION

ACTION A_GetDriveRef:
(* get reference from NC *)
fbAdsRead(
	NETID	:= sIPCNetID,
	PORT	:= AMSPORT_R0_NC,
	IDXGRP	:= NCIDXG_AXPARMS + Axis.NcToPlc.AxisId,
	IDXOFFS	:= NCIDXO_AXP_HWAMSADDR,
	LEN		:= SIZEOF(readBuffer) ,
	DESTADDR:= ADR(readBuffer),
	READ	:= TRUE,
	TMOUT	:= tTimeout
);

IF NOT fbAdsRead.BUSY THEN
	fbAdsRead(READ := FALSE);
	stDriveDiag.nNCAxisID := Axis.NcToPlc.AxisId;

	IF NOT fbAdsRead.ERR THEN
		MEMCPY(ADR(nIds), ADR(readBuffer), SIZEOF(nIds)); 											(* readBuffer[0..5] *)
		MEMCPY(ADR(stDriveRef.nSlaveAddr), ADR(readBuffer[6]), SIZEOF(stDriveRef.nSlaveAddr));  	(* readBuffer[6..7] *)
		MEMCPY(ADR(stDriveRef.nDriveNo), ADR(readBuffer[8]), SIZEOF(stDriveRef.nDriveNo));  		(* readBuffer[8..9] *)

		(* create string out of byte array *)
		stDriveRef.sNetId := F_CreateAmsNetId(nIds);
		bGetDriveRef := FALSE;
	END_IF

	bBusy	:= FALSE;
	iState	:= 0;
END_IF
END_ACTION

ACTION A_Reset:
CASE iSubState OF
0:
	IF stDriveDiag.bWcStateError OR stDriveDiag.bC1DError THEN
		IF stDriveDiag.stClass1Diag.bFeedbackError AND bForcePreopBeforeDrvReset THEN
			(* switch to preop before ResetAmplifier - required for some IndraDrive feedback errors *)
			iSubState := 10;
		ELSE
			(* ResetAmplifier *)
			iSubState := iSubState + 1;
		END_IF
	ELSIF stDriveDiag.stEcSlaveStateBits.bError AND bForceStateChgAfterDrvReset THEN
		(* Clear Error *)
		iSubState := 4;
	ELSIF (NOT stDriveDiag.bOperational) OR stDriveDiag.bAxisError OR (stDriveDiag.iAxisErrorCode <> 0) THEN
		(* NC Reset only *)
		iSubState := 6;
	ELSE
		(* reset not required *)
		iSubState	:= 0;
		iState		:= 0;
		bBusy		:= FALSE;
		bResetAct	:= FALSE;
	END_IF

1:	(* ResetAmplifier *)
	fbReset(
		NetId	:= sIPCNetID,
		Execute:= TRUE,
		Timeout:= DEFAULT_ADS_TIMEOUT,
		Axis	:= Axis,
	);
	IF NOT fbReset.Busy THEN
		fbReset(Execute:= FALSE, Axis:= Axis);

		IF NOT fbReset.Error THEN
			IF bLogDriveDiagMsgs THEN
				strLogMsg := CONCAT('Axis ID: ', DWORD_TO_STRING(Axis.NcToPlc.AxisId));
				strLogMsg := CONCAT(strLogMsg, ', Drive Reset');

				(* report message *)
				ADSLOGSTR(msgCtrlMask := ADSLOG_MSGTYPE_ERROR OR ADSLOG_MSGTYPE_LOG,
					msgFmtStr := strLogMsg, strArg:= '');

				strDiagMsgPrev := '';
			END_IF
			iSubState	:= iSubState + 1;
		ELSE
			bError			:= TRUE;
			iAdsErrId		:= fbReset.AdsErrId;
			iSercosErrId	:= fbReset.SercosErrId;
			bBusy			:= FALSE;
			bResetAct		:= FALSE;
			iSubState		:= 0;
			iState			:= 0;
		END_IF
	END_IF

2:	fbDelay(IN:=TRUE, PT:=t#3s);
	IF fbDelay.Q THEN
		fbDelay(IN:=FALSE);
		iSubState	:= iSubState + 1;
	END_IF

3:	fbGetSlaveState (
		sNetId		:= stDriveRef.sNetId,
		nSlaveAddr	:= stDriveRef.nSlaveAddr,
		bExecute	:= TRUE,
		tTimeout	:= DEFAULT_ADS_TIMEOUT,
	);

	IF NOT fbGetSlaveState.bBusy THEN
		fbGetSlaveState(bExecute:= FALSE);

		IF NOT fbGetSlaveState.bError THEN
			IF ((fbGetSlaveState.state.deviceState <> 16#08) OR ((fbGetSlaveState.state.deviceState AND 16#10) = 16#10)) AND
				bForceStateChgAfterDrvReset THEN

				iSubState	:= iSubState + 1;
			ELSIF Axis.NcToPlc.StateDWord.31 OR (Axis.NcToPlc.ErrorCode <> 0) THEN
				iSubState	:= 6;
			ELSE
				bBusy		:= FALSE;
				bResetAct	:= FALSE;
				iSubState	:= 0;
				iState		:= 0;
			END_IF
		ELSE
			bError			:= TRUE;
			iAdsErrId		:= UDINT_TO_UINT(fbGetSlaveState.nErrId);
			bBusy			:= FALSE;
			bResetAct		:= FALSE;
			iSubState		:= 0;
			iState			:= 0;
		END_IF
	END_IF


(* errors that require CLEAR_ERROR state *)
4:	(* clear error *)
	fbReqSlaveState(
		sNetId		:= stDriveRef.sNetId,
		nSlaveAddr	:= stDriveRef.nSlaveAddr,
		bExecute	:= TRUE,
		tTimeout	:= DEFAULT_ADS_TIMEOUT,
		state		:= EC_DEVICE_STATE_ERROR);

	IF NOT fbReqSlaveState.bBusy THEN
		fbReqSlaveState(bExecute:= FALSE);

		IF NOT fbReqSlaveState.bError THEN
			iSubState	:= iSubState + 1;
		ELSE
			bError		:= TRUE;
			iAdsErrId	:= UDINT_TO_UINT(fbReqSlaveState.nErrId);
			bBusy		:= FALSE;
			bResetAct	:= FALSE;
			iSubState	:= 0;
			iState		:= 0;
		END_IF
	END_IF

5:	(* set op *)
	fbReqSlaveState(
		sNetId		:= stDriveRef.sNetId,
		nSlaveAddr	:= stDriveRef.nSlaveAddr,
		bExecute	:= TRUE,
		tTimeout	:= DEFAULT_ADS_TIMEOUT,
		state		:= EC_DEVICE_STATE_OP);

	IF NOT fbReqSlaveState.bBusy THEN
		fbReqSlaveState(bExecute:= FALSE);

		IF NOT fbReqSlaveState.bError THEN
			iSubState	:= iSubState + 1;
		ELSE
			bError		:= TRUE;
			iAdsErrId	:= UDINT_TO_UINT(fbReqSlaveState.nErrId);
			bBusy		:= FALSE;
			bResetAct	:= FALSE;
			iSubState	:= 0;
			iState		:= 0;
		END_IF
	END_IF

6:	fbNcReset(
		Execute:= TRUE,
		Axis:= Axis,
	);

	IF fbNcReset.Done OR fbNcReset.Error THEN
		IF fbNcReset.Error THEN
			bError 		:= TRUE;
			iAdsErrId 	:= UDINT_TO_UINT(fbNcReset.ErrorID);
		END_IF

		iSubState	:= 0;
		iState		:= 0;
		bBusy		:= FALSE;
		bResetAct	:= FALSE;
		fbNcReset(Execute:= FALSE, Axis:= Axis);
	END_IF


(* errors that only can be reset if in PREOP (parameter mode) *)
10:	(* set preop *)
	fbReqSlaveState(
		sNetId		:= stDriveRef.sNetId,
		nSlaveAddr	:= stDriveRef.nSlaveAddr,
		bExecute	:= TRUE,
		tTimeout	:= DEFAULT_ADS_TIMEOUT,
		state		:= EC_DEVICE_STATE_PREOP);

	IF NOT fbReqSlaveState.bBusy THEN
		fbReqSlaveState(bExecute:= FALSE);

		IF NOT fbReqSlaveState.bError THEN
			iSubState	:= iSubState + 1;
		ELSE
			bError		:= TRUE;
			iAdsErrId	:= UDINT_TO_UINT(fbReqSlaveState.nErrId);
			bBusy		:= FALSE;
			bResetAct	:= FALSE;
			iSubState	:= 0;
			iState		:= 0;
		END_IF
	END_IF

11:	(* ResetAmplifier *)
	fbReset(
		NetId	:= sIPCNetID,
		Execute:= TRUE,
		Timeout:= DEFAULT_ADS_TIMEOUT,
		Axis	:= Axis,
	);
	IF NOT fbReset.Busy THEN
		fbReset(Execute:= FALSE, Axis:= Axis);

		IF NOT fbReset.Error THEN
			IF bLogDriveDiagMsgs THEN
				strLogMsg := CONCAT('Axis ID: ', DWORD_TO_STRING(Axis.NcToPlc.AxisId));
				strLogMsg := CONCAT(strLogMsg, ', Drive Reset');

				(* report message *)
				ADSLOGSTR(msgCtrlMask := ADSLOG_MSGTYPE_ERROR OR ADSLOG_MSGTYPE_LOG,
					msgFmtStr := strLogMsg, strArg:= '');

				strDiagMsgPrev := '';
			END_IF
			iSubState	:= iSubState + 1;
		ELSE
			bError			:= TRUE;
			iAdsErrId		:= fbReset.AdsErrId;
			iSercosErrId	:= fbReset.SercosErrId;
			bBusy			:= FALSE;
			bResetAct		:= FALSE;
			iSubState		:= 0;
			iState			:= 0;
		END_IF
	END_IF

12:	fbDelay(IN:=TRUE, PT:=t#3s);
	IF fbDelay.Q THEN
		fbDelay(IN:=FALSE);
		iSubState	:= iSubState + 1;
	END_IF

13:	(* set op *)
	fbReqSlaveState(
		sNetId		:= stDriveRef.sNetId,
		nSlaveAddr	:= stDriveRef.nSlaveAddr,
		bExecute	:= TRUE,
		tTimeout	:= DEFAULT_ADS_TIMEOUT,
		state		:= EC_DEVICE_STATE_OP);

	IF NOT fbReqSlaveState.bBusy THEN
		fbReqSlaveState(bExecute:= FALSE);

		IF NOT fbReqSlaveState.bError THEN
			iSubState	:= iSubState + 1;
		ELSE
			bError		:= TRUE;
			iAdsErrId	:= UDINT_TO_UINT(fbReqSlaveState.nErrId);
			bBusy		:= FALSE;
			bResetAct	:= FALSE;
			iSubState	:= 0;
			iState		:= 0;
		END_IF
	END_IF

14:	(* ResetAmplifier *)
	fbReset(
		NetId	:= sIPCNetID,
		Execute:= TRUE,
		Timeout:= DEFAULT_ADS_TIMEOUT,
		Axis	:= Axis,
	);
	IF NOT fbReset.Busy THEN
		fbReset(Execute:= FALSE, Axis:= Axis);

		IF NOT fbReset.Error THEN
			IF bLogDriveDiagMsgs THEN
				strLogMsg := CONCAT('Axis ID: ', DWORD_TO_STRING(Axis.NcToPlc.AxisId));
				strLogMsg := CONCAT(strLogMsg, ', Drive Reset');

				(* report message *)
				ADSLOGSTR(msgCtrlMask := ADSLOG_MSGTYPE_ERROR OR ADSLOG_MSGTYPE_LOG,
					msgFmtStr := strLogMsg, strArg:= '');

				strDiagMsgPrev := '';
			END_IF
			iSubState	:= iSubState + 1;
		ELSE
			bError			:= TRUE;
			iAdsErrId		:= fbReset.AdsErrId;
			iSercosErrId	:= fbReset.SercosErrId;
			bBusy			:= FALSE;
			bResetAct		:= FALSE;
			iSubState		:= 0;
			iState			:= 0;
		END_IF
	END_IF

15:	fbDelay(IN:=TRUE, PT:=t#3s);
	IF fbDelay.Q THEN
		fbDelay(IN:=FALSE);
		iSubState	:= iSubState + 1;
	END_IF

16:	fbNcReset(
		Execute:= TRUE,
		Axis:= Axis,
	);

	IF fbNcReset.Done OR fbNcReset.Error THEN
		IF fbNcReset.Error THEN
			bError 		:= TRUE;
			iAdsErrId 	:= UDINT_TO_UINT(fbNcReset.ErrorID);
		END_IF

		iSubState	:= 0;
		iState		:= 0;
		bBusy		:= FALSE;
		bResetAct	:= FALSE;
		fbNcReset(Execute:= FALSE, Axis:= Axis);
	END_IF

END_CASE
END_ACTION

END_FUNCTION_BLOCK

// Motion/MotionCore/FB_MC2AXIS
FUNCTION_BLOCK FB_MC2AXIS
VAR_INPUT
	/// AmsNetId of the IPC 
	IPCNetID: T_AmsNetId := '';
	eAxisType: E_AxisType := E_AxisType.AX5xxx;
	eEncoderType: E_EncoderType := E_EncoderType.Resolver;
	///	Power auf Achse	
	bEnableAxis: BOOL;
	///	Limit switch positiv		
	bEnablePos: BOOL;
	///	Limit switch negativ	
	bEnableNeg: BOOL;
	///	Referenzschalter	
	bCalibrationCam: BOOL;
	///	Override für alle Bewegungen	
	fOverride: LREAL := 100;
	///	Drehmomentbegrenzung	
	fMaxMom: REAL := 100.0;
	FloatingCmd: ST_FloatingCmd;
	///	Reset Cmd	
	bReset: BOOL;
	///	Externer Diagnose Request	
	bDiagReq: BOOL;
	///	Commandos und Positionen	
	ToMc2: ST_ToMc2;
	///	setzt Done Flag auf FALSE	
	bClear: BOOL;
	///	stellt die beim Ausschalten gesicherte Position wieder ein	
	bRestorePosAfterRestart: BOOL := TRUE;
END_VAR
VAR_OUTPUT
	bError: BOOL;
	FromMc2: ST_FromMc2;
	bDone: BOOL;
	bInitOk: BOOL;
	/// contains sNetID of EcMaster, nSlaveAddr of EcDrive, nDriveNo of EcDrive, either preset or read from NC 
	DriveRef: ST_DriveRef;
END_VAR
VAR
	bLockPosPers: BOOL;
	diCmdCounter: UDINT;
	posDone: R_TRIG;
	bRestart: BOOL;
	bMovementCmd: BOOL;
	bResetReq: BOOL;
	bEcStateOk: BOOL;
	///	axis reference data structure 	
	srctAxis: AXIS_REF;
	IiCurrentTourque AT %I*: INT;
	QiTourqueMax AT %Q*: INT;
	Iui_MotTemp AT %I*: UINT;
	EcState AT %I*: WORD;
	fbPowerAxis: MC_Power;
	///	Power function block output data 			
	PowerAxisOut: ST_McOutputs;
	HomeAxis: MC_Home;
	///	Home function block output data			
	HomeOut: ST_McOutputs;
	MoveAbsAxis1: MC_MoveAbsolute;
	MoveAbsAxis2: MC_MoveAbsolute;
	///	Move abs function block output data 		
	MoveAbsOut1: ST_McOutputs;
	MoveAbsOut2: ST_McOutputs;
	MoveRelAxis1: MC_MoveRelative;
	MoveRelAxis2: MC_MoveRelative;
	///	Move rel function block output data		
	MoveRelOut1: ST_McOutputs;
	MoveRelOut2: ST_McOutputs;
	MoveAddAxis1: MC_MoveAdditive;
	MoveAddAxis2: MC_MoveAdditive;
	///	Move Additive function block output data		
	MoveAddOut1: ST_McOutputs;
	MoveAddOut2: ST_McOutputs;
	MoveModAxis: MC_MoveModulo;
	///	Move abs function block output data 		
	MoveModOut: ST_McOutputs;
	MoveVelAxis1: MC_MoveVelocity;
	MoveVelAxis2: MC_MoveVelocity;
	///	Move abs function block output data 		
	MoveVelOut1: ST_McOutputs;
	MoveVelOut2: ST_McOutputs;
	JogAxis: MC_Jog;
	///	Jog function block output data			
	JogOut: ST_McOutputs;
	StopAxis: MC_Stop;
	///	Stop function block output data			
	StopOut: ST_McOutputs;
	HaltAxis: MC_Halt;
	///	Halt function block output data			
	HaltOut: ST_McOutputs;
	SetPosition: MC_SetPosition;
	///	Halt function block output data			
	SetPositionOut: ST_McOutputs;
	enState: E_Mc2AxisState;
	///	AX5000	
	/// axes diag + reset 
	fbAxisDiag: FB_AX5000Diag;
	stAX5000Diag: ST_AX5000Diag;
	bDiagAct: BOOL;
	///	AX2000, EL72..		
	fbResetAxis: MC_Reset;
	fPosTmp: REAL;
	fbResetAxisFloating: MC_Reset;
	tonResetFloating: TON;
	fbFloatingAbsAxis1: MC_MoveAbsolute;
	fbFloatingAbsAxis2: MC_MoveAbsolute;
	fbFloatingMoveTrig: FB_TON_RMTH;
	///	Reset function block output data 			
	ResetOut: ST_McOutputs;
	diTest: DINT;
	bJogForward: BOOL;
	bJogBackwards: BOOL;
	posResetErr: R_TRIG;
	ton_StartDelay: TON;
	iStepResetPosPers: INT;
	bFederOffReset: BOOL;
	fIstPosPers: REAL;
END_VAR

(*
	Default axis function block
	www.rmth.at / 2008

	Version 1:	Thomas Pavelec
	Version 2: 	Roland Ertl

***************************************************************)
(* update the axis status at the beginning of each cycle *)
srctAxis.ReadStatus( );

DriveRef := fbAxisDiag.DriveRef;

bEcStateOk := (EcState = 8) OR (eAxisType = Virtual OR eAxisType = DigIO);
ton_StartDelay(PT := T#4s);
IF (srctAxis.Status.NcCycleCounter > 0) AND bEcStateOk THEN	(*	NOT srctAxis.Status.DriveDeviceError	*)
	ton_StartDelay.IN := TRUE;
END_IF

(*	IInit + restore + save position if no abs encoder...	*)(*	IInit + restore + save position if no abs encoder...	*)
IF NOT bInitOk THEN
	FromMc2.sStatusText := 'Axis Init NOK';
	IF NOT bError AND ton_StartDelay.Q THEN
		(*	no Abs multi turn	*)
		IF eEncoderType <> MultiTurnAbs AND bRestorePosAfterRestart THEN
			IF NOT HomeAxis.Execute OR HomeAxis.Error THEN
				HomeAxis(Execute := FALSE , Axis:=srctAxis);
			END_IF
			HomeAxis.Position := fIstPosPers;
			HomeAxis.HomingMode := MC_Direct;
			HomeAxis.Options.ClearPositionLag := TRUE;
			HomeAxis(Execute := TRUE ,  Axis:=srctAxis);

			bLockPosPers := FALSE;
			bInitOk := HomeAxis.Done AND NOT HomeAxis.Error;
		ELSE
			bLockPosPers := FALSE;
			bInitOk := TRUE;
		END_IF
	ELSE
		FromMc2.sStatusText := 'Axis not ready';
		(*	make reset possible because of  one cable feedback error	*)
		IF (ToMc2.Command = Mc2CmdReset OR bReset) THEN
			bResetReq := TRUE;
		END_IF
	END_IF

(*	INIT OK	*)
ELSE
	FromMc2.sStatusText := 'Axis ready';
	IF bEcStateOk THEN
		IF NOT bLockPosPers THEN
			fIstPosPers := FromMc2.fActPos;	(*	save last position	*)
		ELSE
			FromMc2.sStatusText := 'Pos Pers locked';
		END_IF
	ELSE
		FromMc2.sStatusText := 'EC State NOK';
		bLockPosPers := TRUE;
	END_IF
END_IF

(*	Position latch error reset	*)
IF bLockPosPers AND bInitOk THEN
	(*	reset	*)
	CASE iStepResetPosPers OF

		0:
			IF bError AND (ToMc2.Command = Mc2CmdReset OR bReset) AND ton_StartDelay.Q THEN
				iStepResetPosPers := 10;
				HomeAxis(Execute := FALSE ,  Axis:=srctAxis);
			END_IF

		10:
			bResetReq := TRUE;
			iStepResetPosPers := 11;

		11:
			IF ResetOut.Done AND NOT ResetOut.Error THEN
				bResetReq := FALSE;
				iStepResetPosPers := 20;
			ELSIF ResetOut.Error THEN
				iStepResetPosPers := 0;
			END_IF

		20:
			HomeAxis.Position := fIstPosPers;
			HomeAxis.HomingMode := MC_Direct;
			HomeAxis.Options.ClearPositionLag := TRUE;
			HomeAxis(Execute := TRUE ,  Axis:=srctAxis);
			IF HomeAxis.Done AND NOT HomeAxis.Error THEN
				HomeAxis(Execute := FALSE ,  Axis:=srctAxis);
				iStepResetPosPers := 100;
			ELSIF HomeAxis.Error THEN
				iStepResetPosPers := 0;
			END_IF

		100:
			bLockPosPers := FALSE;
			iStepResetPosPers := 0;

	END_CASE
ELSE
	iStepResetPosPers := 0;
END_IF

(* Diag + Reset *)
A_Tourque( );
A_AxisDiag( );

IF (ToMc2.Command = Mc2CmdReset OR bReset) AND bInitOk THEN
	enState := Mc2AxisStateReset;
END_IF

IF bInitOk THEN
	CASE enState OF
		Mc2AxisStateInit:
			(* initialisation *)
			(* initialize all function blocks *)
			bResetReq := FALSE;
			bMovementCmd := FALSE;
			A_ResMovExecute();
			StopAxis.Execute := FALSE;
			HaltAxis.Execute := FALSE;
			SetPosition.Execute := FALSE;
			enState := Mc2AxisStateIdle;

	(*	wait for new job	*)
		Mc2AxisStateIdle:
			(*	reset	*)
			IF MoveAbsAxis1.Active  OR NOT MoveAbsAxis1.Busy THEN
				MoveAbsAxis1.Execute := FALSE;
			END_IF;
			IF MoveAbsAxis2.Active  OR NOT MoveAbsAxis2.Busy THEN
				MoveAbsAxis2.Execute := FALSE;
			END_IF;
			IF MoveRelAxis1.Active  OR NOT MoveRelAxis1.Busy THEN
				MoveRelAxis1.Execute := FALSE;
			END_IF;
			IF MoveRelAxis2.Active  OR NOT MoveRelAxis2.Busy THEN
				MoveRelAxis2.Execute := FALSE;
			END_IF;
			IF MoveAddAxis1.Active  OR NOT MoveAddAxis1.Busy THEN
				MoveAddAxis1.Execute := FALSE;
			END_IF;
			IF MoveAddAxis2.Active  OR NOT MoveAddAxis2.Busy THEN
				MoveAddAxis2.Execute := FALSE;
			END_IF;
			IF MoveVelAxis1.Active  OR NOT MoveVelAxis1.Busy THEN
				MoveVelAxis1.Execute := FALSE;
			END_IF;
			IF MoveVelAxis2.Active  OR NOT MoveVelAxis2.Busy THEN
				MoveVelAxis2.Execute := FALSE;
			END_IF;
			(*	clear done flag	*)
			IF bClear THEN
				bClear := FALSE;
				bDone := FALSE;
			END_IF
			(*	check for new job	*)
			A_GetCommand( );

		Mc2AxisStateHome:
			bMovementCmd := FALSE;
			A_ResMovExecute();
			HomeAxis.Position := ToMc2.strctHomPrm.Position;
			HomeAxis.HomingMode := ToMc2.strctHomPrm.HomingMode;
			HomeAxis.BufferMode := ToMc2.strctHomPrm.BufferMode;
			HomeAxis.bCalibrationCam := bCalibrationCam;
			HomeAxis.Execute := TRUE;
			IF HomeAxis.Done THEN
				bDone := TRUE;
				bInitOk := TRUE;
				HomeAxis.Execute := FALSE;
				ToMc2.Command := Mc2CmdNothing;
				enState := Mc2AxisStateIdle;
			ELSIF HomeAxis.Error THEN
				FromMc2.nErrorId := HomeAxis.ErrorID;
				FromMc2.sErrorSource := 'MC_Home';
				enState := Mc2AxisStateError;
			ELSE
				A_GetCommand();
			END_IF

		Mc2AxisStateSetPos:
			bMovementCmd := FALSE;
			A_ResMovExecute();
			SetPosition.Position := ToMc2.strctSetPosPrm.Position;
			SetPosition.Mode := ToMc2.strctSetPosPrm.Mode;
			SetPosition.Options.ClearPositionLag := ToMc2.strctSetPosPrm.ClearPositionLag;
			SetPosition.Execute := TRUE;
			IF SetPosition.Done THEN
				bDone := TRUE;
				SetPosition.Execute := FALSE;
				ToMc2.Command := Mc2CmdNothing;
				enState := Mc2AxisStateIdle;
			ELSIF SetPosition.Error THEN
				FromMc2.nErrorId := SetPosition.ErrorID;
				FromMc2.sErrorSource := 'MC_SetPosition';
				enState := Mc2AxisStateError;
			ELSE
				A_GetCommand();
			END_IF

		Mc2AxisStateJog:
			bMovementCmd := FALSE;
			bRestart := (bJogBackwards <> ToMc2.strctJogPrm.JogBackwards) OR
						(bJogForward <> ToMc2.strctJogPrm.JogForward)  OR
						(JogAxis.Mode <> ToMc2.strctJogPrm.Mode) OR
						(JogAxis.Velocity <> ToMc2.strctJogPrm.Velocity);
			JogAxis.Mode := ToMc2.strctJogPrm.Mode;
			JogAxis.Position := ToMc2.strctJogPrm.Position;
			JogAxis.Velocity := ToMc2.strctJogPrm.Velocity;
			JogAxis.Acceleration := ToMc2.strctJogPrm.Acceleration;
			JogAxis.Deceleration := ToMc2.strctJogPrm.Deceleration;
			JogAxis.Jerk := ToMc2.strctJogPrm.Jerk;
			bJogBackwards := ToMc2.strctJogPrm.JogBackwards;
			bJogForward := ToMc2.strctJogPrm.JogForward;
			IF bRestart THEN
				JogAxis.JogBackwards:=FALSE;
				JogAxis.JogForward:=FALSE;
			ELSE
				JogAxis.JogBackwards:=bJogBackwards;
				JogAxis.JogForward:=bJogForward;
			END_IF
			bDone := FALSE;
			IF JogAxis.Error THEN
				FromMc2.nErrorId := JogAxis.ErrorID;
				FromMc2.sErrorSource := 'MC_Jog';
				enState := Mc2AxisStateError;
			END_IF

			A_GetCommand();

		Mc2AxisStateHalt:
			(* HALT ist zu bevorzugen gegenüber STOP -> Schnellstopp *)
			bMovementCmd := FALSE;
			A_ResMovExecute();
			HaltAxis.Deceleration := ToMc2.strctMovPrm.Deceleration;
			HaltAxis.Jerk := ToMc2.strctMovPrm.Jerk;
			HaltAxis.BufferMode := ToMc2.strctMovPrm.BufferMode;
			HaltAxis.Execute := TRUE;
			StopAxis.Execute := FALSE;
			SetPosition.Execute := FALSE;
			IF HaltAxis.Done THEN
				bDone := TRUE;
				ToMc2.Command := Mc2CmdNothing;
				HaltAxis.Execute := FALSE;
				enState := Mc2AxisStateIdle;
			ELSIF HaltAxis.Error THEN
				FromMc2.nErrorId := HaltAxis.ErrorID;
				FromMc2.sErrorSource := 'MC_Halt';
				enState := Mc2AxisStateError;
			END_IF

		Mc2AxisStateStop:
			bMovementCmd := FALSE;
			A_ResMovExecute();
			StopAxis.Deceleration := ToMc2.strctMovPrm.Deceleration;
			StopAxis.Jerk := ToMc2.strctMovPrm.Jerk;
			StopAxis.Execute := TRUE;
			HaltAxis.Execute := FALSE;
			SetPosition.Execute := FALSE;
			IF StopAxis.Done THEN
				bDone := TRUE;
				(*	ToMc2.Command := Mc2CmdNothing;
					StopAxis.Execute := FALSE;		*)
				(*	enState := Mc2AxisStateIdle;	*)
				A_GetCommand( );
			ELSIF StopAxis.Error THEN
				FromMc2.nErrorId := StopAxis.ErrorID;
				FromMc2.sErrorSource := 'MC_Stop';
				enState := Mc2AxisStateError;
			END_IF

		Mc2AxisStateMovAbs:
			bMovementCmd := TRUE;
			(* FB1 bevorzugen *)
			(* Busy ist high, wenn ein Befehl ansteht; Active ist high, wenn der Mov-Befehl ausgeführt wird *)
			IF NOT MoveAbsAxis1.Busy THEN
				MoveAbsAxis1.Position := ToMc2.strctMovPrm.Position;
				MoveAbsAxis1.Velocity := ToMc2.strctMovPrm.Velocity;
				MoveAbsAxis1.Acceleration := ToMc2.strctMovPrm.Acceleration;
				MoveAbsAxis1.Deceleration := ToMc2.strctMovPrm.Deceleration;
				MoveAbsAxis1.Jerk := ToMc2.strctMovPrm.Jerk;
				MoveAbsAxis1.BufferMode := ToMc2.strctMovPrm.BufferMode;
				MoveAbsAxis1(Execute := TRUE , Axis:=srctAxis);
				IF MoveAbsAxis1.Error THEN
					FromMc2.nErrorId := MoveAbsAxis1.ErrorID;
					FromMc2.sErrorSource := 'MC_MoveAbsolute1';
					enState := Mc2AxisStateError;
				ELSE
					ToMc2.Command := Mc2CmdNothing;
					enState := Mc2AxisStateIdle;
				END_IF
			ELSIF NOT MoveAbsAxis2.Busy THEN
				MoveAbsAxis2.Position := ToMc2.strctMovPrm.Position;
				MoveAbsAxis2.Velocity := ToMc2.strctMovPrm.Velocity;
				MoveAbsAxis2.Acceleration := ToMc2.strctMovPrm.Acceleration;
				MoveAbsAxis2.Deceleration := ToMc2.strctMovPrm.Deceleration;
				MoveAbsAxis2.Jerk := ToMc2.strctMovPrm.Jerk;
				MoveAbsAxis2.BufferMode := ToMc2.strctMovPrm.BufferMode;
				MoveAbsAxis2(Execute := TRUE , Axis:=srctAxis);
				IF MoveAbsAxis2.Error THEN
					FromMc2.nErrorId := MoveAbsAxis2.ErrorID;
					FromMc2.sErrorSource := 'MC_MoveAbsolute2';
					enState := Mc2AxisStateError;
				ELSE
					ToMc2.Command := Mc2CmdNothing;
					enState := Mc2AxisStateIdle;
				END_IF
			END_IF

		Mc2AxisStateMovRel:
			bMovementCmd := TRUE;
			IF ToMc2.strctMovPrm.Direction = MC_Positive_Direction THEN
				fPosTmp := ToMc2.strctMovPrm.Position;
			ELSE
				fPosTmp := - ToMc2.strctMovPrm.Position;
			END_IF

			(* FB1 bevorzugen *)
			(* Busy ist high, wenn ein Befehl ansteht; Active ist high, wenn der Mov-Befehl ausgeführt wird *)
			IF NOT MoveRelAxis1.Busy THEN
				MoveRelAxis1.Distance := fPosTmp;
				MoveRelAxis1.Velocity := ToMc2.strctMovPrm.Velocity;
				MoveRelAxis1.Acceleration := ToMc2.strctMovPrm.Acceleration;
				MoveRelAxis1.Deceleration := ToMc2.strctMovPrm.Deceleration;
				MoveRelAxis1.Jerk := ToMc2.strctMovPrm.Jerk;
				MoveRelAxis1.BufferMode := ToMc2.strctMovPrm.BufferMode;
				MoveRelAxis1(Execute := TRUE , Axis:=srctAxis);
				IF MoveRelAxis1.Error THEN
					FromMc2.nErrorId := MoveRelAxis1.ErrorID;
					FromMc2.sErrorSource := 'MC_MoveRelative1';
					enState := Mc2AxisStateError;
				ELSE
					ToMc2.Command := Mc2CmdNothing;
					enState := Mc2AxisStateIdle;
				END_IF;
			(* wenn FB1 aktiv -> neues Kommando mit FB2 überlagern *)
			ELSIF NOT MoveRelAxis2.Busy THEN
				MoveRelAxis2.Distance := fPosTmp;
				MoveRelAxis2.Velocity := ToMc2.strctMovPrm.Velocity;
				MoveRelAxis2.Acceleration := ToMc2.strctMovPrm.Acceleration;
				MoveRelAxis2.Deceleration := ToMc2.strctMovPrm.Deceleration;
				MoveRelAxis2.Jerk := ToMc2.strctMovPrm.Jerk;
				MoveRelAxis2.BufferMode := ToMc2.strctMovPrm.BufferMode;
				MoveRelAxis2(Execute := TRUE , Axis:=srctAxis);
				IF MoveRelAxis2.Error THEN
					FromMc2.nErrorId := MoveRelAxis2.ErrorID;
					FromMc2.sErrorSource := 'MC_MoveRelative2';
					enState := Mc2AxisStateError;
				ELSE
					ToMc2.Command := Mc2CmdNothing;
					enState := Mc2AxisStateIdle;
				END_IF;
			END_IF;


		Mc2AxisStateMovAdd:
			bMovementCmd := TRUE;
			IF ToMc2.strctMovPrm.Direction = MC_Positive_Direction THEN
				fPosTmp := ToMc2.strctMovPrm.Position;
			ELSE
				fPosTmp := - ToMc2.strctMovPrm.Position;
			END_IF

			(* FB1 bevorzugen *)
			(* Busy ist high, wenn ein Befehl ansteht; Active ist high, wenn der Mov-Befehl ausgeführt wird *)
			IF NOT MoveAddAxis1.Busy THEN
				MoveAddAxis1.Distance := fPosTmp;
				MoveAddAxis1.Velocity := ToMc2.strctMovPrm.Velocity;
				MoveAddAxis1.Acceleration := ToMc2.strctMovPrm.Acceleration;
				MoveAddAxis1.Deceleration := ToMc2.strctMovPrm.Deceleration;
				MoveAddAxis1.Jerk := ToMc2.strctMovPrm.Jerk;
				MoveAddAxis1.BufferMode := ToMc2.strctMovPrm.BufferMode;
				MoveAddAxis1(Execute := TRUE , Axis:=srctAxis);
				IF MoveAddAxis1.Error THEN
					FromMc2.nErrorId := MoveAddAxis1.ErrorID;
					FromMc2.sErrorSource := 'MC_MoveAdditive1';
					enState := Mc2AxisStateError;
				ELSE
					ToMc2.Command := Mc2CmdNothing;
					enState := Mc2AxisStateIdle;
				END_IF
			(* wenn FB1 aktiv -> neues Kommando mit FB2 überlagern *)
			ELSIF NOT MoveAddAxis2.Busy THEN
				MoveAddAxis2.Distance := fPosTmp;
				MoveAddAxis2.Velocity := ToMc2.strctMovPrm.Velocity;
				MoveAddAxis2.Acceleration := ToMc2.strctMovPrm.Acceleration;
				MoveAddAxis2.Deceleration := ToMc2.strctMovPrm.Deceleration;
				MoveAddAxis2.Jerk := ToMc2.strctMovPrm.Jerk;
				MoveAddAxis2.BufferMode := ToMc2.strctMovPrm.BufferMode;
				MoveAddAxis2(Execute := TRUE , Axis:=srctAxis);
				IF MoveAddAxis2.Error THEN
					FromMc2.nErrorId := MoveAddAxis2.ErrorID;
					FromMc2.sErrorSource := 'MC_MoveAdditive2';
					enState := Mc2AxisStateError;
				ELSE
					ToMc2.Command := Mc2CmdNothing;
					enState := Mc2AxisStateIdle;
				END_IF
			END_IF

		Mc2AxisStateMovMod:
			bMovementCmd := TRUE;
			MoveModAxis.Position := ToMc2.strctMovPrm.Position;
			MoveModAxis.Velocity := ToMc2.strctMovPrm.Velocity;
			MoveModAxis.Acceleration := ToMc2.strctMovPrm.Acceleration;
			MoveModAxis.Deceleration := ToMc2.strctMovPrm.Deceleration;
			MoveModAxis.Jerk := ToMc2.strctMovPrm.Jerk;
			MoveModAxis.BufferMode := ToMc2.strctMovPrm.BufferMode;
			MoveModAxis.Direction := ToMc2.strctMovPrm.Direction;
			MoveModAxis(Execute := TRUE , Axis:=srctAxis);
			IF MoveModAxis.Active  THEN
				ToMc2.Command := Mc2CmdNothing;
				MoveModAxis.Execute := FALSE;
				enState := Mc2AxisStateIdle;
			ELSIF MoveModAxis.Error THEN
				FromMc2.nErrorId := MoveModAxis.ErrorID;
				FromMc2.sErrorSource := 'MC_MoveModulo';
				enState := Mc2AxisStateError;
			ELSE
				A_GetCommand();
			END_IF

		Mc2AxisStateMovVel:
			bMovementCmd := TRUE;
			(* FB1 bevorzugen *)
			(* Busy ist high, wenn ein Befehl ansteht; Active ist high, wenn der Mov-Befehl ausgeführt wird *)
			IF NOT MoveVelAxis1.Busy THEN
				MoveVelAxis1.Velocity := ToMc2.strctMovPrm.Velocity;
				MoveVelAxis1.Acceleration := ToMc2.strctMovPrm.Acceleration;
				MoveVelAxis1.Deceleration := ToMc2.strctMovPrm.Deceleration;
				MoveVelAxis1.Jerk := ToMc2.strctMovPrm.Jerk;
				MoveVelAxis1.BufferMode := ToMc2.strctMovPrm.BufferMode;
				MoveVelAxis1.Direction := ToMc2.strctMovPrm.Direction;
				MoveVelAxis1(Execute := TRUE , Axis:=srctAxis);
				IF MoveVelAxis1.Error THEN
					FromMc2.nErrorId := MoveVelAxis1.ErrorID;
					FromMc2.sErrorSource := 'MC_MoveVelocity1';
					enState := Mc2AxisStateError;
				ELSE
					ToMc2.Command := Mc2CmdNothing;
					enState := Mc2AxisStateIdle;
				END_IF
			(* wenn FB1 aktiv -> neues Kommando mit FB2 überlagern *)
			ELSIF NOT MoveVelAxis2.Busy THEN
				MoveVelAxis2.Velocity := ToMc2.strctMovPrm.Velocity;
				MoveVelAxis2.Acceleration := ToMc2.strctMovPrm.Acceleration;
				MoveVelAxis2.Deceleration := ToMc2.strctMovPrm.Deceleration;
				MoveVelAxis2.Jerk := ToMc2.strctMovPrm.Jerk;
				MoveVelAxis2.BufferMode := ToMc2.strctMovPrm.BufferMode;
				MoveVelAxis2.Direction := ToMc2.strctMovPrm.Direction;
				MoveVelAxis2(Execute := TRUE , Axis:=srctAxis);
				IF MoveVelAxis2.Error THEN
					FromMc2.nErrorId := MoveVelAxis2.ErrorID;
					FromMc2.sErrorSource := 'MC_MoveVelocity2';
					enState := Mc2AxisStateError;
				ELSE
					ToMc2.Command := Mc2CmdNothing;
					enState := Mc2AxisStateIdle;
				END_IF
			END_IF;

		Mc2AxisStateError:
			bMovementCmd := FALSE;
			FromMc2.bError := TRUE;
			HaltAxis.Execute := TRUE;

		Mc2AxisStateReset:
			bMovementCmd := FALSE;
			bResetReq := TRUE;
			HaltAxis.Execute := FALSE;
			diTest := diTest + 1;
			IF ResetOut.Done THEN
				bReset := FALSE;
				bResetReq := FALSE;
				ToMc2.Command := Mc2CmdNothing;
				FromMc2.bError := FALSE;
				FromMc2.nErrorId := 0;
				FromMc2.sErrorSource := '';
				enState := Mc2AxisStateInit;
			ELSIF posResetErr.Q THEN
				bReset := FALSE;
				bResetReq := FALSE;
				FromMc2.bError := TRUE;
				FromMc2.nErrorId := fbAxisDiag.AdsErrId;
				FromMc2.sErrorSource := 'MC_Reset';
			END_IF

	END_CASE
END_IF

A_Halt( );			(* call the halt function block			 		*)
A_Home( );		(* call the home function block			 	*)
A_Jog( );			(* call the jog function block			 		*)
A_Power( );		(* call the power function block			 	*)
A_MovRel( );		(* call the move relative function block 		*)
A_MovAdd( );		(* call the move additive function block 		*)
A_MovAbs( );		(* call the move absolute function block 		*)
A_MovMod( );		(* call the move modulo function block 		*)
A_MovVel( );		(* call the move velo function block 		*)
A_Stop( );		(* call the stop function block			 		*)
A_SetPosition( );	(* call the set position function block 		*)

srctAxis.ReadStatus( );

IF srctAxis.Status.Error THEN
	FromMc2.bError := TRUE;
END_IF

bError := FromMc2.bError OR srctAxis.Status.Error OR bLockPosPers;
FromMc2.bNotMoving := srctAxis.NcToPlc.StateDWord.2;
FromMc2.bReady := srctAxis.NcToPlc.StateDWord.0 AND NOT srctAxis.NcToPlc.StateDWord.31 AND NOT bLockPosPers;	(*	Ready and no error	*)
FromMc2.InTargetPosition := srctAxis.Status.InTargetPosition AND FromMc2.bNotMoving;
FromMc2.bCoupled:= srctAxis.Status.Coupled;
FromMc2.nAxisId :=srctAxis.NcToPlc.AxisId;

FromMc2.fActPos := srctAxis.NcToPlc.ActPos;
FromMc2.fActModPos := srctAxis.NcToPlc.ModuloActPos;
FromMc2.fActVelo := srctAxis.NcToPlc.ActVelo;
FromMc2.bMovesPos := AxisIsMovingForward(srctAxis.NcToPlc.StateDWord);
FromMc2.bMovesNeg := AxisIsMovingBackwards(srctAxis.NcToPlc.StateDWord);
FromMc2.bHasJob := AxisHasJob( srctAxis.NcToPlc.StateDWord );
FromMc2.bEnabled := fbPowerAxis.Enable AND NOT srctAxis.Status.Disabled AND srctAxis.Status.Operational;

(**)
posDone(CLK := MoveAbsAxis1.Done OR MoveAbsAxis2.Done OR
				MoveRelAxis1.Done OR MoveRelAxis2.Done OR
				MoveModAxis.Done OR
				MoveAddAxis1.Done OR MoveAddAxis2.Done OR
				MoveVelAxis1.InVelocity OR MoveVelAxis2.InVelocity);

(*	MoveAbsAxis.Done	*)
IF bMovementCmd THEN
	IF posDone.Q THEN
		bDone := TRUE;
	END_IF
END_IF

(*	Ausgabe allg. Achsfehler	*)
IF bError AND FromMc2.nErrorId=0 AND FromMc2.sErrorSource='' THEN
	FromMc2.nErrorId:=srctAxis.NcToPlc.ErrorCode;
	FromMc2.sErrorSource:='srctAxis';
END_IF;

FromMc2.AxisState := enState;

FromMc2.PowerAxisOut := PowerAxisOut;
FromMc2.ResetOut := ResetOut;
FromMc2.HomeOut := HomeOut;

(* Move abs out Kombination und einzeln *)
IF MoveAbsOut1.Busy OR NOT MoveAbsOut2.Busy THEN
	FromMc2.MoveAbsOut := MoveAbsOut1;
ELSE
	FromMc2.MoveAbsOut := MoveAbsOut2;
END_IF;
FromMc2.MoveAbsOut1 := MoveAbsOut1;
FromMc2.MoveAbsOut2 := MoveAbsOut2;

(* Move rel out Kombination und einzeln *)
IF MoveRelOut1.Busy OR NOT MoveRelOut2.Busy THEN
	FromMc2.MoveRelOut := MoveRelOut1;
ELSE
	FromMc2.MoveRelOut := MoveRelOut2;
END_IF;
FromMc2.MoveRelOut1 := MoveRelOut1;
FromMc2.MoveRelOut2 := MoveRelOut2;

(* MOVE add out Kombination und einzeln *)
IF MoveAddOut1.Busy OR NOT MoveAddOut2.Busy THEN
	FromMc2.MoveAddOut := MoveAddOut1;
ELSE
	FromMc2.MoveAddOut := MoveAddOut2;
END_IF;
FromMc2.MoveAddOut1 := MoveAddOut1;
FromMc2.MoveAddOut2 := MoveAddOut2;

(* MOVE add out Kombination und einzeln *)
IF MoveVelOut1.Busy OR NOT MoveVelOut2.Busy THEN
	FromMc2.MoveVelOut := MoveVelOut1;
ELSE
	FromMc2.MoveVelOut := MoveVelOut2;
END_IF;
FromMc2.MoveVelOut1 := MoveVelOut1;
FromMc2.MoveVelOut2 := MoveVelOut2;

FromMc2.JogOut := JogOut;
FromMc2.MoveModOut := MoveModOut;
FromMc2.StopOut := StopOut;
FromMc2.HaltOut := HaltOut;

ToMc2.Command := Mc2CmdNothing;

ACTION A_AxisDiag:
(* clear active flags for reset/diag *)
bDiagAct := FALSE;

(*	reset servo hardware	*)
IF eAxisType = AX5xxx THEN
	(* Diag + Reset of AX5000 *)
	(* call drive diag FBs *)
	fbAxisDiag(
		IPCNetID	:= IPCNetID,
		Axis		:= srctAxis,
		stAX5000Diag:= stAX5000Diag,
		Reset   	:= bResetReq,
		GetDiag 	:= bDiagReq
	);
	
	(* update active flags for reset/diag *)
	ResetOut.Done := fbAxisDiag.ResetDone;
	ResetOut.Active := fbAxisDiag.ResetAct;
	ResetOut.Busy := fbAxisDiag.Busy;
	ResetOut.Error := fbAxisDiag.Error;
	ResetOut.ErrorID := fbAxisDiag.AdsErrId;

	bDiagAct	:= fbAxisDiag.DiagAct;

	(* clear reset/diag request if not active *)
	bResetReq		:= bResetReq AND ResetOut.Active;
	bDiagReq		:= bDiagReq AND bDiagAct;

(*	only reset NC	*)
ELSIF eAxisType = EL72xx OR eAxisType = AX2xxx OR eAxisType = Virtual OR eAxisType = DigIO OR eAxisType = Lenze_94xx THEN
	fbResetAxis(
		Execute:= bResetReq,
		Axis:= srctAxis,
		Done=> ResetOut.Done,
		Busy=> ResetOut.Busy,
		Error=> ResetOut.Error,
		ErrorID=> ResetOut.ErrorID);
	IF fbResetAxis.Done THEN
		bResetReq := FALSE;
	END_IF

ELSE
	;
END_IF

posResetErr(CLK := ResetOut.Error);
END_ACTION

ACTION A_GetCommand:
(*	get command action	*)

IF enState = Mc2AxisStateError THEN
	RETURN;
END_IF

IF ToMc2.Command = Mc2CmdHalt THEN
	enState := Mc2AxisStateHalt;
	bDone := FALSE;

ELSIF ToMc2.Command = Mc2CmdStop THEN
	enState := Mc2AxisStateStop;
	bDone := FALSE;

ELSIF ToMc2.Command = Mc2CmdHome THEN
	enState := Mc2AxisStateHome;
	bDone := FALSE;
	diCmdCounter := diCmdCounter + 1;

ELSIF ToMc2.Command = Mc2CmdMovAbs THEN
	enState := Mc2AxisStateMovAbs;
	bDone := FALSE;
	diCmdCounter := diCmdCounter + 1;

ELSIF ToMc2.Command = Mc2CmdMovRel THEN
	enState := Mc2AxisStateMovRel;
	bDone := FALSE;
	diCmdCounter := diCmdCounter + 1;

ELSIF ToMc2.Command = Mc2CmdMovAdd THEN
	enState := Mc2AxisStateMovAdd;
	bDone := FALSE;
	diCmdCounter := diCmdCounter + 1;

ELSIF ToMc2.Command = Mc2CmdMovMod THEN
	enState := Mc2AxisStateMovMod;
	bDone := FALSE;
	diCmdCounter := diCmdCounter + 1;

ELSIF ToMc2.Command = Mc2CmdMovVel THEN
	enState := Mc2AxisStateMovVel;
	bDone := FALSE;
	diCmdCounter := diCmdCounter + 1;

ELSIF ToMc2.Command = Mc2CmdJog OR (ToMc2.strctJogPrm.JogForward OR ToMc2.strctJogPrm.JogBackwards) THEN
	IF FromMc2.bNotMoving AND NOT srctAxis.Status.HasJob THEN
		enState := Mc2AxisStateJog;
	END_IF

ELSIF ToMc2.Command = Mc2CmdSetPos THEN
	enState := Mc2AxisStateSetPos;
	bDone := FALSE;

END_IF
END_ACTION

ACTION A_Halt:
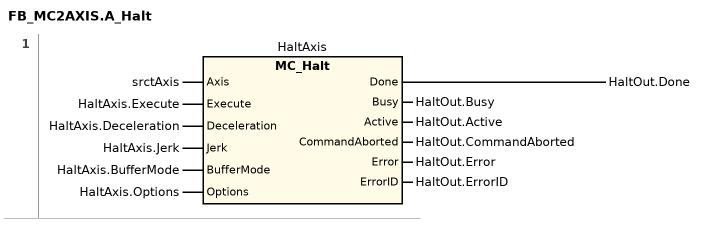
// NETWORK 1
HaltAxis(
    Axis := srctAxis,
    Execute := HaltAxis.Execute,
    Deceleration := HaltAxis.Deceleration,
    Jerk := HaltAxis.Jerk,
    BufferMode := HaltAxis.BufferMode,
    Options := HaltAxis.Options,
    Busy => HaltOut.Busy,
    Active => HaltOut.Active,
    CommandAborted => HaltOut.CommandAborted,
    Error => HaltOut.Error,
    ErrorID => HaltOut.ErrorID); // MC_Halt
HaltOut.Done := HaltAxis.Done;
END_ACTION

